LIN {X 0,Y 474.292,Z 613.364,A -85,B 0,C 180,E1 -7469.284,E2 -7469.284} C_VEL
LIN {X 0,Y 475.962,Z 468.165,A -85,B 0,C 180,E1 -7471.57,E2 -7471.57} C_VEL
LIN {X 0,Y 471.306,Z 449.007,A -85,B 0,C 180,E1 -7472.133,E2 -7472.133} C_VEL
LIN {X 0,Y 471.034,Z 448.055,A -85,B 0,C 180,E1 -7472.181,E2 -7472.181} C_VEL
LIN {X 0,Y 469.089,Z 439.057,A -85,B 0,C 180,E1 -7473.866,E2 -7473.866} C_VEL
LIN {X 0,Y 467.706,Z 432.847,A -85,B 0,C 180,E1 -7475.065,E2 -7475.065} C_VEL
LIN {X 0,Y 467.699,Z 432.856,A -85,B 0,C 180,E1 -7477.773,E2 -7477.773} C_VEL
LIN {X 0,Y 467.676,Z 432.847,A -85,B 0,C 180,E1 -7481.266,E2 -7481.266} C_VEL
LIN {X 0,Y 467.615,Z 432.864,A -85,B 0,C 180,E1 -7483.915,E2 -7483.915} C_VEL
LIN {X 0,Y 467.6,Z 432.861,A -85,B 0,C 180,E1 -7486.593,E2 -7486.593} C_VEL
LIN {X 0,Y 467.628,Z 432.861,A -85,B 0,C 180,E1 -7489.308,E2 -7489.308} C_VEL
LIN {X 0,Y 467.541,Z 432.872,A -85,B 0,C 180,E1 -7492.074,E2 -7492.074} C_VEL
LIN {X 0,Y 467.608,Z 432.856,A -85,B 0,C 180,E1 -7494.887,E2 -7494.887} C_VEL
LIN {X 0,Y 467.631,Z 432.857,A -85,B 0,C 180,E1 -7497.768,E2 -7497.768} C_VEL
LIN {X 0,Y 467.573,Z 432.865,A -85,B 0,C 180,E1 -7501.045,E2 -7501.045} C_VEL
LIN {X 0,Y 467.593,Z 432.863,A -85,B 0,C 180,E1 -7504.242,E2 -7504.242} C_VEL
LIN {X 0,Y 467.553,Z 432.866,A -85,B 0,C 180,E1 -7507.187,E2 -7507.187} C_VEL
LIN {X 0,Y 467.582,Z 432.863,A -85,B 0,C 180,E1 -7510.264,E2 -7510.264} C_VEL
LIN {X 0,Y 467.589,Z 432.858,A -85,B 0,C 180,E1 -7512.567,E2 -7512.567} C_VEL
LIN {X 0,Y 467.573,Z 432.863,A -85,B 0,C 180,E1 -7515.053,E2 -7515.053} C_VEL
LIN {X 0,Y 467.591,Z 432.866,A -85,B 0,C 180,E1 -7517.44,E2 -7517.44} C_VEL
LIN {X 0,Y 467.602,Z 432.86,A -85,B 0,C 180,E1 -7520.857,E2 -7520.857} C_VEL
LIN {X 0,Y 467.565,Z 432.86,A -85,B 0,C 180,E1 -7524.26,E2 -7524.26} C_VEL
LIN {X 0,Y 467.583,Z 432.865,A -85,B 0,C 180,E1 -7527.321,E2 -7527.321} C_VEL
LIN {X 0,Y 467.571,Z 432.857,A -85,B 0,C 180,E1 -7530.667,E2 -7530.667} C_VEL
LIN {X 0,Y 467.629,Z 432.858,A -85,B 0,C 180,E1 -7533.2,E2 -7533.2} C_VEL
LIN {X 0,Y 467.593,Z 432.852,A -85,B 0,C 180,E1 -7536.468,E2 -7536.468} C_VEL
LIN {X 0,Y 467.623,Z 432.863,A -85,B 0,C 180,E1 -7539.777,E2 -7539.777} C_VEL
LIN {X 0,Y 467.609,Z 432.853,A -85,B 0,C 180,E1 -7542.507,E2 -7542.507} C_VEL
LIN {X 0,Y 467.606,Z 432.857,A -85,B 0,C 180,E1 -7545.196,E2 -7545.196} C_VEL
LIN {X 0,Y 467.656,Z 432.855,A -85,B 0,C 180,E1 -7547.854,E2 -7547.854} C_VEL
LIN {X 0,Y 467.682,Z 432.845,A -85,B 0,C 180,E1 -7551.357,E2 -7551.357} C_VEL
LIN {X 0,Y 467.743,Z 432.845,A -85,B 0,C 180,E1 -7553.962,E2 -7553.962} C_VEL
LIN {X 0,Y 467.859,Z 432.824,A -85,B 0,C 180,E1 -7557.417,E2 -7557.417} C_VEL
LIN {X 0,Y 467.882,Z 432.829,A -85,B 0,C 180,E1 -7560,E2 -7560} C_VEL
LIN {X 0,Y 467.86,Z 432.824,A -85,B 0,C 180,E1 -7562.583,E2 -7562.583} C_VEL
LIN {X 0,Y 467.743,Z 432.843,A -85,B 0,C 180,E1 -7566.037,E2 -7566.037} C_VEL
LIN {X 0,Y 467.681,Z 432.849,A -85,B 0,C 180,E1 -7568.643,E2 -7568.643} C_VEL
LIN {X 0,Y 467.655,Z 432.848,A -85,B 0,C 180,E1 -7572.145,E2 -7572.145} C_VEL
LIN {X 0,Y 467.639,Z 432.862,A -85,B 0,C 180,E1 -7575.695,E2 -7575.695} C_VEL
LIN {X 0,Y 467.616,Z 432.849,A -85,B 0,C 180,E1 -7578.764,E2 -7578.764} C_VEL
LIN {X 0,Y 467.58,Z 432.864,A -85,B 0,C 180,E1 -7581.268,E2 -7581.268} C_VEL
LIN {X 0,Y 467.573,Z 432.868,A -85,B 0,C 180,E1 -7583.943,E2 -7583.943} C_VEL
LIN {X 0,Y 467.615,Z 432.858,A -85,B 0,C 180,E1 -7586.8,E2 -7586.8} C_VEL
LIN {X 0,Y 467.579,Z 432.87,A -85,B 0,C 180,E1 -7589.736,E2 -7589.736} C_VEL
LIN {X 0,Y 467.583,Z 432.862,A -85,B 0,C 180,E1 -7592.758,E2 -7592.758} C_VEL
LIN {X 0,Y 467.556,Z 432.871,A -85,B 0,C 180,E1 -7595.889,E2 -7595.889} C_VEL
LIN {X 0,Y 467.582,Z 432.864,A -85,B 0,C 180,E1 -7599.145,E2 -7599.145} C_VEL
LIN {X 0,Y 467.586,Z 432.862,A -85,B 0,C 180,E1 -7602.567,E2 -7602.567} C_VEL
LIN {X 0,Y 467.57,Z 432.865,A -85,B 0,C 180,E1 -7605.053,E2 -7605.053} C_VEL
LIN {X 0,Y 467.625,Z 432.862,A -85,B 0,C 180,E1 -7607.444,E2 -7607.444} C_VEL
LIN {X 0,Y 467.582,Z 432.864,A -85,B 0,C 180,E1 -7610.855,E2 -7610.855} C_VEL
LIN {X 0,Y 467.56,Z 432.871,A -85,B 0,C 180,E1 -7614.261,E2 -7614.261} C_VEL
LIN {X 0,Y 467.582,Z 432.869,A -85,B 0,C 180,E1 -7617.321,E2 -7617.321} C_VEL
LIN {X 0,Y 467.595,Z 432.887,A -85,B 0,C 180,E1 -7619.549,E2 -7619.549} C_VEL
LIN {X 0,Y 471.189,Z 447.756,A -85,B 0,C 180,E1 -7622.098,E2 -7622.098} C_VEL
LIN {X 0,Y 472.292,Z 452.989,A -85,B 0,C 180,E1 -7622.963,E2 -7622.963} C_VEL
LIN {X 0,Y 471.349,Z 470.678,A -85,B 0,C 180,E1 -7625.577,E2 -7625.577} C_VEL
LIN {X 0,Y 471.209,Z 472.852,A -85,B 0,C 180,E1 -7625.88,E2 -7625.88} C_VEL
LIN {X 0,Y 475.856,Z 496.892,A -85,B 0,C 180,E1 -7626.517,E2 -7626.517} C_VEL
LIN {X 0,Y 474.168,Z 638.503,A -85,B 0,C 180,E1 -7628.736,E2 -7628.736} C_VEL
LIN {X 0,Y 473.646,Z 654.003,A -85,B 0,C 180,E1 -7629.138,E2 -7629.138} C_VEL
LIN {X 0,Y 473.017,Z 668.829,A -85,B 0,C 180,E1 -7629.7,E2 -7629.7} C_VEL
LIN {X 0,Y 472.245,Z 683.472,A -85,B 0,C 180,E1 -7630.437,E2 -7630.437} C_VEL
LIN {X 0,Y 471.45,Z 697.08,A -85,B 0,C 180,E1 -7631.306,E2 -7631.306} C_VEL
LIN {X 0,Y 470.626,Z 709.613,A -85,B 0,C 180,E1 -7632.286,E2 -7632.286} C_VEL
LIN {X 0,Y 469.805,Z 722.347,A -85,B 0,C 180,E1 -7633.487,E2 -7633.487} C_VEL
LIN {X 0,Y 468.951,Z 733.908,A -85,B 0,C 180,E1 -7634.795,E2 -7634.795} C_VEL
LIN {X 0,Y 468.346,Z 743.643,A -85,B 0,C 180,E1 -7636.107,E2 -7636.107} C_VEL
LIN {X 0,Y 467.661,Z 753.221,A -85,B 0,C 180,E1 -7637.639,E2 -7637.639} C_VEL
LIN {X 0,Y 467.377,Z 761.161,A -85,B 0,C 180,E1 -7639.166,E2 -7639.166} C_VEL
LIN {X 0,Y 467.011,Z 768.591,A -85,B 0,C 180,E1 -7640.908,E2 -7640.908} C_VEL
LIN {X 0,Y 466.818,Z 774.485,A -85,B 0,C 180,E1 -7642.647,E2 -7642.647} C_VEL
LIN {X 0,Y 466.721,Z 777.986,A -85,B 0,C 180,E1 -7643.949,E2 -7643.949} C_VEL
LIN {X 0,Y 466.616,Z 781.525,A -85,B 0,C 180,E1 -7645.681,E2 -7645.681} C_VEL
LIN {X 0,Y 466.638,Z 783.854,A -85,B 0,C 180,E1 -7647.41,E2 -7647.41} C_VEL
LIN {X 0,Y 466.616,Z 785.022,A -85,B 0,C 180,E1 -7649.137,E2 -7649.137} C_VEL
LIN {X 0,Y 466.615,Z 785.016,A -85,B 0,C 180,E1 -7650.863,E2 -7650.863} C_VEL
LIN {X 0,Y 466.64,Z 783.835,A -85,B 0,C 180,E1 -7652.589,E2 -7652.589} C_VEL
LIN {X 0,Y 466.616,Z 781.496,A -85,B 0,C 180,E1 -7654.318,E2 -7654.318} C_VEL
LIN {X 0,Y 466.73,Z 777.954,A -85,B 0,C 180,E1 -7656.05,E2 -7656.05} C_VEL
LIN {X 0,Y 466.834,Z 773.112,A -85,B 0,C 180,E1 -7657.786,E2 -7657.786} C_VEL
LIN {X 0,Y 467.053,Z 766.845,A -85,B 0,C 180,E1 -7659.527,E2 -7659.527} C_VEL
LIN {X 0,Y 467.518,Z 758.98,A -85,B 0,C 180,E1 -7661.269,E2 -7661.269} C_VEL
LIN {X 0,Y 467.904,Z 750.519,A -85,B 0,C 180,E1 -7662.814,E2 -7662.814} C_VEL
LIN {X 0,Y 468.512,Z 740.532,A -85,B 0,C 180,E1 -7664.33,E2 -7664.33} C_VEL
LIN {X 0,Y 469.197,Z 730.234,A -85,B 0,C 180,E1 -7665.641,E2 -7665.641} C_VEL
LIN {X 0,Y 469.997,Z 718.835,A -85,B 0,C 180,E1 -7666.862,E2 -7666.862} C_VEL
LIN {X 0,Y 470.742,Z 706.933,A -85,B 0,C 180,E1 -7667.933,E2 -7667.933} C_VEL
LIN {X 0,Y 471.619,Z 693.812,A -85,B 0,C 180,E1 -7668.911,E2 -7668.911} C_VEL
LIN {X 0,Y 472.463,Z 679.406,A -85,B 0,C 180,E1 -7669.779,E2 -7669.779} C_VEL
LIN {X 0,Y 473.21,Z 665.055,A -85,B 0,C 180,E1 -7670.453,E2 -7670.453} C_VEL
LIN {X 0,Y 473.758,Z 650.356,A -85,B 0,C 180,E1 -7670.97,E2 -7670.97} C_VEL
LIN {X 0,Y 474.21,Z 635.624,A -85,B 0,C 180,E1 -7671.318,E2 -7671.318} C_VEL
LIN {X 0,Y 475.906,Z 497.322,A -85,B 0,C 180,E1 -7673.48,E2 -7673.48} C_VEL
LIN {X 0,Y 471.18,Z 472.312,A -85,B 0,C 180,E1 -7674.158,E2 -7674.158} C_VEL
LIN {X 0,Y 472.251,Z 452.84,A -85,B 0,C 180,E1 -7677.036,E2 -7677.036} C_VEL
LIN {X 0,Y 469.543,Z 440.542,A -85,B 0,C 180,E1 -7679.104,E2 -7679.104} C_VEL
LIN {X 0,Y 467.59,Z 432.868,A -85,B 0,C 180,E1 -7680.481,E2 -7680.481} C_VEL
LIN {X 0,Y 467.583,Z 432.865,A -85,B 0,C 180,E1 -7683.787,E2 -7683.787} C_VEL
LIN {X 0,Y 467.547,Z 432.867,A -85,B 0,C 180,E1 -7687.186,E2 -7687.186} C_VEL
LIN {X 0,Y 467.593,Z 432.863,A -85,B 0,C 180,E1 -7690.262,E2 -7690.262} C_VEL
LIN {X 0,Y 467.614,Z 432.859,A -85,B 0,C 180,E1 -7692.571,E2 -7692.571} C_VEL
LIN {X 0,Y 467.565,Z 432.867,A -85,B 0,C 180,E1 -7695.053,E2 -7695.053} C_VEL
LIN {X 0,Y 467.583,Z 432.861,A -85,B 0,C 180,E1 -7697.439,E2 -7697.439} C_VEL
LIN {X 0,Y 467.576,Z 432.866,A -85,B 0,C 180,E1 -7700.855,E2 -7700.855} C_VEL
LIN {X 0,Y 467.557,Z 432.87,A -85,B 0,C 180,E1 -7704.26,E2 -7704.26} C_VEL
LIN {X 0,Y 467.575,Z 432.861,A -85,B 0,C 180,E1 -7707.32,E2 -7707.32} C_VEL
LIN {X 0,Y 467.563,Z 432.869,A -85,B 0,C 180,E1 -7710.667,E2 -7710.667} C_VEL
LIN {X 0,Y 467.62,Z 432.855,A -85,B 0,C 180,E1 -7713.2,E2 -7713.2} C_VEL
LIN {X 0,Y 467.585,Z 432.865,A -85,B 0,C 180,E1 -7716.468,E2 -7716.468} C_VEL
LIN {X 0,Y 467.616,Z 432.857,A -85,B 0,C 180,E1 -7719.777,E2 -7719.777} C_VEL
LIN {X 0,Y 467.602,Z 432.861,A -85,B 0,C 180,E1 -7722.507,E2 -7722.507} C_VEL
LIN {X 0,Y 467.598,Z 432.86,A -85,B 0,C 180,E1 -7725.196,E2 -7725.196} C_VEL
LIN {X 0,Y 467.675,Z 432.851,A -85,B 0,C 180,E1 -7727.855,E2 -7727.855} C_VEL
LIN {X 0,Y 467.675,Z 432.85,A -85,B 0,C 180,E1 -7731.357,E2 -7731.357} C_VEL
LIN {X 0,Y 467.736,Z 432.845,A -85,B 0,C 180,E1 -7733.963,E2 -7733.963} C_VEL
LIN {X 0,Y 467.854,Z 432.826,A -85,B 0,C 180,E1 -7737.417,E2 -7737.417} C_VEL
LIN {X 0,Y 467.875,Z 432.829,A -85,B 0,C 180,E1 -7740,E2 -7740} C_VEL
LIN {X 0,Y 467.854,Z 432.834,A -85,B 0,C 180,E1 -7742.583,E2 -7742.583} C_VEL
LIN {X 0,Y 467.738,Z 432.845,A -85,B 0,C 180,E1 -7746.038,E2 -7746.038} C_VEL
LIN {X 0,Y 467.675,Z 432.856,A -85,B 0,C 180,E1 -7748.643,E2 -7748.643} C_VEL
LIN {X 0,Y 467.648,Z 432.857,A -85,B 0,C 180,E1 -7752.146,E2 -7752.146} C_VEL
LIN {X 0,Y 467.648,Z 432.855,A -85,B 0,C 180,E1 -7755.695,E2 -7755.695} C_VEL
LIN {X 0,Y 467.611,Z 432.862,A -85,B 0,C 180,E1 -7758.765,E2 -7758.765} C_VEL
LIN {X 0,Y 467.575,Z 432.863,A -85,B 0,C 180,E1 -7761.269,E2 -7761.269} C_VEL
LIN {X 0,Y 467.567,Z 432.868,A -85,B 0,C 180,E1 -7763.944,E2 -7763.944} C_VEL
LIN {X 0,Y 467.622,Z 432.86,A -85,B 0,C 180,E1 -7766.8,E2 -7766.8} C_VEL
LIN {X 0,Y 467.582,Z 432.863,A -85,B 0,C 180,E1 -7769.736,E2 -7769.736} C_VEL
LIN {X 0,Y 467.579,Z 432.865,A -85,B 0,C 180,E1 -7772.759,E2 -7772.759} C_VEL
LIN {X 0,Y 467.553,Z 432.871,A -85,B 0,C 180,E1 -7775.89,E2 -7775.89} C_VEL
LIN {X 0,Y 467.615,Z 432.865,A -85,B 0,C 180,E1 -7779.142,E2 -7779.142} C_VEL
LIN {X 0,Y 467.631,Z 432.96,A -85,B 0,C 180,E1 -7780.945,E2 -7780.945} C_VEL
LIN {X 0,Y 470.519,Z 445.746,A -85,B 0,C 180,E1 -7783.4,E2 -7783.4} C_VEL
LIN {X 0,Y 471.119,Z 448.459,A -85,B 0,C 180,E1 -7783.911,E2 -7783.911} C_VEL
LIN {X 0,Y 474.437,Z 461.432,A -85,B 0,C 180,E1 -7784.311,E2 -7784.311} C_VEL
LIN {X 0,Y 476.156,Z 469.425,A -85,B 0,C 180,E1 -7784.534,E2 -7784.534} C_VEL
LIN {X 0,Y 474.316,Z 613.801,A -85,B 0,C 180,E1 -7786.807,E2 -7786.807} C_VEL
LIN {X 0,Y 473.816,Z 629.451,A -85,B 0,C 180,E1 -7787.231,E2 -7787.231} C_VEL
LIN {X 0,Y 473.277,Z 643.627,A -85,B 0,C 180,E1 -7787.784,E2 -7787.784} C_VEL
LIN {X 0,Y 472.516,Z 658.62,A -85,B 0,C 180,E1 -7788.558,E2 -7788.558} C_VEL
LIN {X 0,Y 471.701,Z 672.281,A -85,B 0,C 180,E1 -7789.453,E2 -7789.453} C_VEL
LIN {X 0,Y 471.315,Z 678.799,A -85,B 0,C 180,E1 -7789.955,E2 -7789.955} C_VEL
LIN {X 0,Y 470.421,Z 683.716,A -85,B 0,C 180,E1 -7790.339,E2 -7790.339} C_VEL
LIN {X 0,Y 467.106,Z 691.605,A -85,B 0,C 180,E1 -7790.955,E2 -7790.955} C_VEL
LIN {X 0,Y 463.735,Z 699.161,A -85,B 0,C 180,E1 -7791.631,E2 -7791.631} C_VEL
LIN {X 0,Y 462.763,Z 703.515,A -85,B 0,C 180,E1 -7792.105,E2 -7792.105} C_VEL
LIN {X 0,Y 461.998,Z 713.096,A -85,B 0,C 180,E1 -7793.34,E2 -7793.34} C_VEL
LIN {X 0,Y 461.327,Z 722.98,A -85,B 0,C 180,E1 -7794.85,E2 -7794.85} C_VEL
LIN {X 0,Y 460.739,Z 731.593,A -85,B 0,C 180,E1 -7796.432,E2 -7796.432} C_VEL
LIN {X 0,Y 460.203,Z 739.522,A -85,B 0,C 180,E1 -7798.207,E2 -7798.207} C_VEL
LIN {X 0,Y 459.976,Z 745.004,A -85,B 0,C 180,E1 -7799.722,E2 -7799.722} C_VEL
LIN {X 0,Y 459.74,Z 749.421,A -85,B 0,C 180,E1 -7801.215,E2 -7801.215} C_VEL
LIN {X 0,Y 459.622,Z 752.795,A -85,B 0,C 180,E1 -7802.696,E2 -7802.696} C_VEL
LIN {X 0,Y 459.459,Z 755.962,A -85,B 0,C 180,E1 -7804.641,E2 -7804.641} C_VEL
LIN {X 0,Y 459.411,Z 757.715,A -85,B 0,C 180,E1 -7806.617,E2 -7806.617} C_VEL
LIN {X 0,Y 459.389,Z 758.052,A -85,B 0,C 180,E1 -7808.46,E2 -7808.46} C_VEL
LIN {X 0,Y 459.447,Z 757.117,A -85,B 0,C 180,E1 -7810.335,E2 -7810.335} C_VEL
LIN {X 0,Y 459.533,Z 754.911,A -85,B 0,C 180,E1 -7812.19,E2 -7812.19} C_VEL
LIN {X 0,Y 459.715,Z 751.415,A -85,B 0,C 180,E1 -7814.028,E2 -7814.028} C_VEL
LIN {X 0,Y 459.88,Z 746.602,A -85,B 0,C 180,E1 -7815.847,E2 -7815.847} C_VEL
LIN {X 0,Y 460.206,Z 740.359,A -85,B 0,C 180,E1 -7817.656,E2 -7817.656} C_VEL
LIN {X 0,Y 460.66,Z 732.532,A -85,B 0,C 180,E1 -7819.452,E2 -7819.452} C_VEL
LIN {X 0,Y 461.197,Z 724.229,A -85,B 0,C 180,E1 -7821.014,E2 -7821.014} C_VEL
LIN {X 0,Y 461.921,Z 714.254,A -85,B 0,C 180,E1 -7822.57,E2 -7822.57} C_VEL
LIN {X 0,Y 462.671,Z 704.091,A -85,B 0,C 180,E1 -7823.897,E2 -7823.897} C_VEL
LIN {X 0,Y 463.549,Z 692.016,A -85,B 0,C 180,E1 -7825.217,E2 -7825.217} C_VEL
LIN {X 0,Y 464.521,Z 678.617,A -85,B 0,C 180,E1 -7826.422,E2 -7826.422} C_VEL
LIN {X 0,Y 465.415,Z 665.239,A -85,B 0,C 180,E1 -7827.404,E2 -7827.404} C_VEL
LIN {X 0,Y 466.207,Z 651.434,A -85,B 0,C 180,E1 -7828.219,E2 -7828.219} C_VEL
LIN {X 0,Y 466.911,Z 636.009,A -85,B 0,C 180,E1 -7828.922,E2 -7828.922} C_VEL
LIN {X 0,Y 467.471,Z 620.257,A -85,B 0,C 180,E1 -7829.435,E2 -7829.435} C_VEL
LIN {X 0,Y 467.799,Z 604.734,A -85,B 0,C 180,E1 -7829.758,E2 -7829.758} C_VEL
LIN {X 0,Y 469.488,Z 469.443,A -85,B 0,C 180,E1 -7831.893,E2 -7831.893} C_VEL
LIN {X 0,Y 465.042,Z 451.21,A -85,B 0,C 180,E1 -7832.441,E2 -7832.441} C_VEL
LIN {X 0,Y 463.945,Z 448.293,A -85,B 0,C 180,E1 -7832.565,E2 -7832.565} C_VEL
LIN {X 0,Y 460.678,Z 433.722,A -85,B 0,C 180,E1 -7835.389,E2 -7835.389} C_VEL
LIN {X 0,Y 460.671,Z 433.73,A -85,B 0,C 180,E1 -7837.892,E2 -7837.892} C_VEL
LIN {X 0,Y 460.635,Z 433.726,A -85,B 0,C 180,E1 -7841.44,E2 -7841.44} C_VEL
LIN {X 0,Y 460.559,Z 433.741,A -85,B 0,C 180,E1 -7844.132,E2 -7844.132} C_VEL
LIN {X 0,Y 460.568,Z 433.738,A -85,B 0,C 180,E1 -7846.854,E2 -7846.854} C_VEL
LIN {X 0,Y 460.573,Z 433.744,A -85,B 0,C 180,E1 -7849.616,E2 -7849.616} C_VEL
LIN {X 0,Y 460.517,Z 433.744,A -85,B 0,C 180,E1 -7852.429,E2 -7852.429} C_VEL
LIN {X 0,Y 460.572,Z 433.742,A -85,B 0,C 180,E1 -7855.802,E2 -7855.802} C_VEL
LIN {X 0,Y 460.559,Z 433.735,A -85,B 0,C 180,E1 -7858.233,E2 -7858.233} C_VEL
LIN {X 0,Y 460.526,Z 433.745,A -85,B 0,C 180,E1 -7861.283,E2 -7861.283} C_VEL
LIN {X 0,Y 460.537,Z 433.74,A -85,B 0,C 180,E1 -7864.506,E2 -7864.506} C_VEL
LIN {X 0,Y 460.531,Z 433.739,A -85,B 0,C 180,E1 -7867.62,E2 -7867.62} C_VEL
LIN {X 0,Y 460.546,Z 433.74,A -85,B 0,C 180,E1 -7870.269,E2 -7870.269} C_VEL
LIN {X 0,Y 460.511,Z 433.743,A -85,B 0,C 180,E1 -7873.374,E2 -7873.374} C_VEL
LIN {X 0,Y 460.502,Z 433.743,A -85,B 0,C 180,E1 -7876.624,E2 -7876.624} C_VEL
LIN {X 0,Y 460.56,Z 433.741,A -85,B 0,C 180,E1 -7879.728,E2 -7879.728} C_VEL
LIN {X 0,Y 460.53,Z 433.738,A -85,B 0,C 180,E1 -7882.519,E2 -7882.519} C_VEL
LIN {X 0,Y 460.551,Z 433.741,A -85,B 0,C 180,E1 -7885.624,E2 -7885.624} C_VEL
LIN {X 0,Y 460.538,Z 433.737,A -85,B 0,C 180,E1 -7888.744,E2 -7888.744} C_VEL
LIN {X 0,Y 460.59,Z 433.734,A -85,B 0,C 180,E1 -7892.252,E2 -7892.252} C_VEL
LIN {X 0,Y 460.56,Z 433.735,A -85,B 0,C 180,E1 -7894.705,E2 -7894.705} C_VEL
LIN {X 0,Y 460.511,Z 433.74,A -85,B 0,C 180,E1 -7897.571,E2 -7897.571} C_VEL
LIN {X 0,Y 460.569,Z 433.736,A -85,B 0,C 180,E1 -7900.384,E2 -7900.384} C_VEL
LIN {X 0,Y 460.566,Z 433.731,A -85,B 0,C 180,E1 -7903.146,E2 -7903.146} C_VEL
LIN {X 0,Y 460.555,Z 433.742,A -85,B 0,C 180,E1 -7905.868,E2 -7905.868} C_VEL
LIN {X 0,Y 460.611,Z 433.727,A -85,B 0,C 180,E1 -7908.559,E2 -7908.559} C_VEL
LIN {X 0,Y 460.695,Z 433.721,A -85,B 0,C 180,E1 -7912.108,E2 -7912.108} C_VEL
LIN {X 0,Y 460.697,Z 433.718,A -85,B 0,C 180,E1 -7914.748,E2 -7914.748} C_VEL
LIN {X 0,Y 460.8,Z 433.703,A -85,B 0,C 180,E1 -7917.377,E2 -7917.377} C_VEL
LIN {X 0,Y 460.853,Z 433.704,A -85,B 0,C 180,E1 -7920,E2 -7920} C_VEL
LIN {X 0,Y 460.824,Z 433.7,A -85,B 0,C 180,E1 -7922.622,E2 -7922.622} C_VEL
LIN {X 0,Y 460.709,Z 433.718,A -85,B 0,C 180,E1 -7926.13,E2 -7926.13} C_VEL
LIN {X 0,Y 460.628,Z 433.728,A -85,B 0,C 180,E1 -7928.776,E2 -7928.776} C_VEL
LIN {X 0,Y 460.613,Z 433.723,A -85,B 0,C 180,E1 -7932.445,E2 -7932.445} C_VEL
LIN {X 0,Y 460.599,Z 433.735,A -85,B 0,C 180,E1 -7935.997,E2 -7935.997} C_VEL
LIN {X 0,Y 460.57,Z 433.727,A -85,B 0,C 180,E1 -7938.902,E2 -7938.902} C_VEL
LIN {X 0,Y 460.515,Z 433.747,A -85,B 0,C 180,E1 -7941.485,E2 -7941.485} C_VEL
LIN {X 0,Y 460.542,Z 433.74,A -85,B 0,C 180,E1 -7944.332,E2 -7944.332} C_VEL
LIN {X 0,Y 460.578,Z 433.737,A -85,B 0,C 180,E1 -7947.243,E2 -7947.243} C_VEL
LIN {X 0,Y 460.521,Z 433.742,A -85,B 0,C 180,E1 -7950.239,E2 -7950.239} C_VEL
LIN {X 0,Y 460.529,Z 433.744,A -85,B 0,C 180,E1 -7953.325,E2 -7953.325} C_VEL
LIN {X 0,Y 460.479,Z 433.747,A -85,B 0,C 180,E1 -7956.529,E2 -7956.529} C_VEL
LIN {X 0,Y 460.557,Z 433.742,A -85,B 0,C 180,E1 -7959.86,E2 -7959.86} C_VEL
LIN {X 0,Y 460.513,Z 433.743,A -85,B 0,C 180,E1 -7962.9,E2 -7962.9} C_VEL
LIN {X 0,Y 460.524,Z 433.747,A -85,B 0,C 180,E1 -7965.829,E2 -7965.829} C_VEL
LIN {X 0,Y 460.535,Z 433.742,A -85,B 0,C 180,E1 -7968.989,E2 -7968.989} C_VEL
LIN {X 0,Y 460.526,Z 433.745,A -85,B 0,C 180,E1 -7971.267,E2 -7971.267} C_VEL
LIN {X 0,Y 460.51,Z 433.748,A -85,B 0,C 180,E1 -7974.554,E2 -7974.554} C_VEL
LIN {X 0,Y 460.532,Z 433.744,A -85,B 0,C 180,E1 -7977.715,E2 -7977.715} C_VEL
LIN {X 0,Y 460.548,Z 433.832,A -85,B 0,C 180,E1 -7979.223,E2 -7979.223} C_VEL
LIN {X 0,Y 464.059,Z 448.047,A -85,B 0,C 180,E1 -7981.713,E2 -7981.713} C_VEL
LIN {X 0,Y 465.493,Z 454.798,A -85,B 0,C 180,E1 -7982.849,E2 -7982.849} C_VEL
LIN {X 0,Y 464.454,Z 472.525,A -85,B 0,C 180,E1 -7985.505,E2 -7985.505} C_VEL
LIN {X 0,Y 469.309,Z 497.459,A -85,B 0,C 180,E1 -7986.184,E2 -7986.184} C_VEL
LIN {X 0,Y 467.541,Z 638.122,A -85,B 0,C 180,E1 -7988.419,E2 -7988.419} C_VEL
LIN {X 0,Y 466.99,Z 653.689,A -85,B 0,C 180,E1 -7988.826,E2 -7988.826} C_VEL
LIN {X 0,Y 466.321,Z 669.079,A -85,B 0,C 180,E1 -7989.419,E2 -7989.419} C_VEL
LIN {X 0,Y 465.537,Z 683.208,A -85,B 0,C 180,E1 -7990.143,E2 -7990.143} C_VEL
LIN {X 0,Y 464.674,Z 696.828,A -85,B 0,C 180,E1 -7991.023,E2 -7991.023} C_VEL
LIN {X 0,Y 463.73,Z 710.667,A -85,B 0,C 180,E1 -7992.127,E2 -7992.127} C_VEL
LIN {X 0,Y 462.858,Z 723.186,A -85,B 0,C 180,E1 -7993.345,E2 -7993.345} C_VEL
LIN {X 0,Y 462.047,Z 733.678,A -85,B 0,C 180,E1 -7994.562,E2 -7994.562} C_VEL
LIN {X 0,Y 461.38,Z 743.417,A -85,B 0,C 180,E1 -7995.893,E2 -7995.893} C_VEL
LIN {X 0,Y 460.783,Z 751.983,A -85,B 0,C 180,E1 -7997.267,E2 -7997.267} C_VEL
LIN {X 0,Y 460.444,Z 759.928,A -85,B 0,C 180,E1 -7998.778,E2 -7998.778} C_VEL
LIN {X 0,Y 459.979,Z 766.687,A -85,B 0,C 180,E1 -8000.324,E2 -8000.324} C_VEL
LIN {X 0,Y 459.776,Z 772.941,A -85,B 0,C 180,E1 -8002.092,E2 -8002.092} C_VEL
LIN {X 0,Y 459.637,Z 777.777,A -85,B 0,C 180,E1 -8003.855,E2 -8003.855} C_VEL
LIN {X 0,Y 459.533,Z 781.317,A -85,B 0,C 180,E1 -8005.614,E2 -8005.614} C_VEL
LIN {X 0,Y 459.56,Z 783.647,A -85,B 0,C 180,E1 -8007.37,E2 -8007.37} C_VEL
LIN {X 0,Y 459.519,Z 784.815,A -85,B 0,C 180,E1 -8009.123,E2 -8009.123} C_VEL
LIN {X 0,Y 459.518,Z 784.809,A -85,B 0,C 180,E1 -8010.876,E2 -8010.876} C_VEL
LIN {X 0,Y 459.563,Z 783.627,A -85,B 0,C 180,E1 -8012.629,E2 -8012.629} C_VEL
LIN {X 0,Y 459.532,Z 781.287,A -85,B 0,C 180,E1 -8014.385,E2 -8014.385} C_VEL
LIN {X 0,Y 459.639,Z 777.742,A -85,B 0,C 180,E1 -8016.144,E2 -8016.144} C_VEL
LIN {X 0,Y 459.775,Z 772.9,A -85,B 0,C 180,E1 -8017.907,E2 -8017.907} C_VEL
LIN {X 0,Y 459.978,Z 766.629,A -85,B 0,C 180,E1 -8019.675,E2 -8019.675} C_VEL
LIN {X 0,Y 460.459,Z 758.761,A -85,B 0,C 180,E1 -8021.444,E2 -8021.444} C_VEL
LIN {X 0,Y 460.898,Z 750.525,A -85,B 0,C 180,E1 -8022.975,E2 -8022.975} C_VEL
LIN {X 0,Y 461.573,Z 740.309,A -85,B 0,C 180,E1 -8024.55,E2 -8024.55} C_VEL
LIN {X 0,Y 462.313,Z 730.008,A -85,B 0,C 180,E1 -8025.88,E2 -8025.88} C_VEL
LIN {X 0,Y 463.236,Z 717.683,A -85,B 0,C 180,E1 -8027.212,E2 -8027.212} C_VEL
LIN {X 0,Y 464.067,Z 705.402,A -85,B 0,C 180,E1 -8028.315,E2 -8028.315} C_VEL
LIN {X 0,Y 464.977,Z 691.994,A -85,B 0,C 180,E1 -8029.307,E2 -8029.307} C_VEL
LIN {X 0,Y 465.905,Z 677.195,A -85,B 0,C 180,E1 -8030.185,E2 -8030.185} C_VEL
LIN {X 0,Y 466.637,Z 662.471,A -85,B 0,C 180,E1 -8030.86,E2 -8030.86} C_VEL
LIN {X 0,Y 467.271,Z 647.421,A -85,B 0,C 180,E1 -8031.361,E2 -8031.361} C_VEL
LIN {X 0,Y 467.674,Z 632.474,A -85,B 0,C 180,E1 -8031.689,E2 -8031.689} C_VEL
LIN {X 0,Y 469.36,Z 497.451,A -85,B 0,C 180,E1 -8033.824,E2 -8033.824} C_VEL
LIN {X 0,Y 464.455,Z 472.084,A -85,B 0,C 180,E1 -8034.536,E2 -8034.536} C_VEL
LIN {X 0,Y 465.432,Z 454.521,A -85,B 0,C 180,E1 -8037.178,E2 -8037.178} C_VEL
LIN {X 0,Y 462.709,Z 442.309,A -85,B 0,C 180,E1 -8039.269,E2 -8039.269} C_VEL
LIN {X 0,Y 460.532,Z 433.747,A -85,B 0,C 180,E1 -8040.808,E2 -8040.808} C_VEL
LIN {X 0,Y 460.526,Z 433.744,A -85,B 0,C 180,E1 -8043.324,E2 -8043.324} C_VEL
LIN {X 0,Y 460.475,Z 433.753,A -85,B 0,C 180,E1 -8046.528,E2 -8046.528} C_VEL
LIN {X 0,Y 460.574,Z 433.737,A -85,B 0,C 180,E1 -8049.857,E2 -8049.857} C_VEL
LIN {X 0,Y 460.537,Z 433.738,A -85,B 0,C 180,E1 -8052.904,E2 -8052.904} C_VEL
LIN {X 0,Y 460.505,Z 433.749,A -85,B 0,C 180,E1 -8055.83,E2 -8055.83} C_VEL
LIN {X 0,Y 460.525,Z 433.743,A -85,B 0,C 180,E1 -8058.988,E2 -8058.988} C_VEL
LIN {X 0,Y 460.52,Z 433.743,A -85,B 0,C 180,E1 -8061.267,E2 -8061.267} C_VEL
LIN {X 0,Y 460.507,Z 433.748,A -85,B 0,C 180,E1 -8064.554,E2 -8064.554} C_VEL
LIN {X 0,Y 460.525,Z 433.741,A -85,B 0,C 180,E1 -8067.715,E2 -8067.715} C_VEL
LIN {X 0,Y 460.533,Z 433.744,A -85,B 0,C 180,E1 -8070.769,E2 -8070.769} C_VEL
LIN {X 0,Y 460.561,Z 433.736,A -85,B 0,C 180,E1 -8073.735,E2 -8073.735} C_VEL
LIN {X 0,Y 460.539,Z 433.744,A -85,B 0,C 180,E1 -8076.624,E2 -8076.624} C_VEL
LIN {X 0,Y 460.544,Z 433.736,A -85,B 0,C 180,E1 -8079.453,E2 -8079.453} C_VEL
LIN {X 0,Y 460.552,Z 433.743,A -85,B 0,C 180,E1 -8082.23,E2 -8082.23} C_VEL
LIN {X 0,Y 460.557,Z 433.738,A -85,B 0,C 180,E1 -8084.965,E2 -8084.965} C_VEL
LIN {X 0,Y 460.622,Z 433.728,A -85,B 0,C 180,E1 -8087.666,E2 -8087.666} C_VEL
LIN {X 0,Y 460.622,Z 433.728,A -85,B 0,C 180,E1 -8091.224,E2 -8091.224} C_VEL
LIN {X 0,Y 460.702,Z 433.72,A -85,B 0,C 180,E1 -8093.87,E2 -8093.87} C_VEL
LIN {X 0,Y 460.819,Z 433.702,A -85,B 0,C 180,E1 -8097.378,E2 -8097.378} C_VEL
LIN {X 0,Y 460.845,Z 433.705,A -85,B 0,C 180,E1 -8100,E2 -8100} C_VEL
LIN {X 0,Y 460.819,Z 433.71,A -85,B 0,C 180,E1 -8102.623,E2 -8102.623} C_VEL
LIN {X 0,Y 460.704,Z 433.722,A -85,B 0,C 180,E1 -8106.13,E2 -8106.13} C_VEL
LIN {X 0,Y 460.622,Z 433.733,A -85,B 0,C 180,E1 -8108.776,E2 -8108.776} C_VEL
LIN {X 0,Y 460.606,Z 433.739,A -85,B 0,C 180,E1 -8112.445,E2 -8112.445} C_VEL
LIN {X 0,Y 460.615,Z 433.734,A -85,B 0,C 180,E1 -8116.008,E2 -8116.008} C_VEL
LIN {X 0,Y 460.563,Z 433.737,A -85,B 0,C 180,E1 -8119.616,E2 -8119.616} C_VEL
LIN {X 0,Y 460.505,Z 433.752,A -85,B 0,C 180,E1 -8122.429,E2 -8122.429} C_VEL
LIN {X 0,Y 460.563,Z 433.74,A -85,B 0,C 180,E1 -8125.803,E2 -8125.803} C_VEL
LIN {X 0,Y 460.553,Z 433.745,A -85,B 0,C 180,E1 -8128.233,E2 -8128.233} C_VEL
LIN {X 0,Y 460.52,Z 433.744,A -85,B 0,C 180,E1 -8131.285,E2 -8131.285} C_VEL
LIN {X 0,Y 460.53,Z 433.745,A -85,B 0,C 180,E1 -8134.507,E2 -8134.507} C_VEL
LIN {X 0,Y 460.527,Z 433.746,A -85,B 0,C 180,E1 -8137.621,E2 -8137.621} C_VEL
LIN {X 0,Y 460.567,Z 433.805,A -85,B 0,C 180,E1 -8140.602,E2 -8140.602} C_VEL
LIN {X 0,Y 463.443,Z 446.216,A -85,B 0,C 180,E1 -8143.033,E2 -8143.033} C_VEL
LIN {X 0,Y 463.962,Z 448.732,A -85,B 0,C 180,E1 -8143.513,E2 -8143.513} C_VEL
LIN {X 0,Y 466.156,Z 454.96,A -85,B 0,C 180,E1 -8143.744,E2 -8143.744} C_VEL
LIN {X 0,Y 469.604,Z 469.923,A -85,B 0,C 180,E1 -8144.188,E2 -8144.188} C_VEL
LIN {X 0,Y 467.734,Z 613.627,A -85,B 0,C 180,E1 -8146.482,E2 -8146.482} C_VEL
LIN {X 0,Y 467.234,Z 629.203,A -85,B 0,C 180,E1 -8146.905,E2 -8146.905} C_VEL
LIN {X 0,Y 466.594,Z 644.62,A -85,B 0,C 180,E1 -8147.518,E2 -8147.518} C_VEL
LIN {X 0,Y 465.82,Z 658.855,A -85,B 0,C 180,E1 -8148.267,E2 -8148.267} C_VEL
LIN {X 0,Y 464.972,Z 672.601,A -85,B 0,C 180,E1 -8149.182,E2 -8149.182} C_VEL
LIN {X 0,Y 464.091,Z 685.353,A -85,B 0,C 180,E1 -8150.223,E2 -8150.223} C_VEL
LIN {X 0,Y 463.227,Z 697.249,A -85,B 0,C 180,E1 -8151.397,E2 -8151.397} C_VEL
LIN {X 0,Y 462.763,Z 703.515,A -85,B 0,C 180,E1 -8152.105,E2 -8152.105} C_VEL
LIN {X 0,Y 461.824,Z 707.77,A -85,B 0,C 180,E1 -8152.6,E2 -8152.6} C_VEL
LIN {X 0,Y 458.551,Z 714.532,A -85,B 0,C 180,E1 -8153.406,E2 -8153.406} C_VEL
LIN {X 0,Y 455.243,Z 720.853,A -85,B 0,C 180,E1 -8154.27,E2 -8154.27} C_VEL
LIN {X 0,Y 454.264,Z 724.419,A -85,B 0,C 180,E1 -8154.852,E2 -8154.852} C_VEL
LIN {X 0,Y 453.68,Z 733.014,A -85,B 0,C 180,E1 -8156.496,E2 -8156.496} C_VEL
LIN {X 0,Y 453.166,Z 740.231,A -85,B 0,C 180,E1 -8158.178,E2 -8158.178} C_VEL
LIN {X 0,Y 452.917,Z 745.604,A -85,B 0,C 180,E1 -8159.715,E2 -8159.715} C_VEL
LIN {X 0,Y 452.649,Z 749.938,A -85,B 0,C 180,E1 -8161.229,E2 -8161.229} C_VEL
LIN {X 0,Y 452.448,Z 754.173,A -85,B 0,C 180,E1 -8163.227,E2 -8163.227} C_VEL
LIN {X 0,Y 452.32,Z 756.88,A -85,B 0,C 180,E1 -8165.197,E2 -8165.197} C_VEL
LIN {X 0,Y 452.29,Z 758.179,A -85,B 0,C 180,E1 -8167.142,E2 -8167.142} C_VEL
LIN {X 0,Y 452.34,Z 758.139,A -85,B 0,C 180,E1 -8169.063,E2 -8169.063} C_VEL
LIN {X 0,Y 452.359,Z 756.798,A -85,B 0,C 180,E1 -8170.959,E2 -8170.959} C_VEL
LIN {X 0,Y 452.467,Z 754.173,A -85,B 0,C 180,E1 -8172.836,E2 -8172.836} C_VEL
LIN {X 0,Y 452.695,Z 750.249,A -85,B 0,C 180,E1 -8174.698,E2 -8174.698} C_VEL
LIN {X 0,Y 452.901,Z 744.997,A -85,B 0,C 180,E1 -8176.541,E2 -8176.541} C_VEL
LIN {X 0,Y 453.205,Z 739.626,A -85,B 0,C 180,E1 -8178.038,E2 -8178.038} C_VEL
LIN {X 0,Y 453.66,Z 732.191,A -85,B 0,C 180,E1 -8179.738,E2 -8179.738} C_VEL
LIN {X 0,Y 454.305,Z 723.67,A -85,B 0,C 180,E1 -8181.34,E2 -8181.34} C_VEL
LIN {X 0,Y 455.064,Z 713.656,A -85,B 0,C 180,E1 -8182.903,E2 -8182.903} C_VEL
LIN {X 0,Y 455.879,Z 703.37,A -85,B 0,C 180,E1 -8184.25,E2 -8184.25} C_VEL
LIN {X 0,Y 456.845,Z 691.066,A -85,B 0,C 180,E1 -8185.589,E2 -8185.589} C_VEL
LIN {X 0,Y 457.797,Z 678.144,A -85,B 0,C 180,E1 -8186.752,E2 -8186.752} C_VEL
LIN {X 0,Y 458.712,Z 665.396,A -85,B 0,C 180,E1 -8187.696,E2 -8187.696} C_VEL
LIN {X 0,Y 459.538,Z 651.573,A -85,B 0,C 180,E1 -8188.522,E2 -8188.522} C_VEL
LIN {X 0,Y 460.23,Z 637.433,A -85,B 0,C 180,E1 -8189.18,E2 -8189.18} C_VEL
LIN {X 0,Y 460.806,Z 622.279,A -85,B 0,C 180,E1 -8189.7,E2 -8189.7} C_VEL
LIN {X 0,Y 461.172,Z 606.382,A -85,B 0,C 180,E1 -8190.055,E2 -8190.055} C_VEL
LIN {X 0,Y 463.026,Z 470.802,A -85,B 0,C 180,E1 -8192.223,E2 -8192.223} C_VEL
LIN {X 0,Y 459.032,Z 454.277,A -85,B 0,C 180,E1 -8192.728,E2 -8192.728} C_VEL
LIN {X 0,Y 456.814,Z 448.521,A -85,B 0,C 180,E1 -8192.961,E2 -8192.961} C_VEL
LIN {X 0,Y 453.647,Z 434.599,A -85,B 0,C 180,E1 -8195.724,E2 -8195.724} C_VEL
LIN {X 0,Y 453.597,Z 434.609,A -85,B 0,C 180,E1 -8198.914,E2 -8198.914} C_VEL
LIN {X 0,Y 453.606,Z 434.607,A -85,B 0,C 180,E1 -8202.551,E2 -8202.551} C_VEL
LIN {X 0,Y 453.549,Z 434.613,A -85,B 0,C 180,E1 -8206.196,E2 -8206.196} C_VEL
LIN {X 0,Y 453.524,Z 434.615,A -85,B 0,C 180,E1 -8209.041,E2 -8209.041} C_VEL
LIN {X 0,Y 453.481,Z 434.625,A -85,B 0,C 180,E1 -8211.836,E2 -8211.836} C_VEL
LIN {X 0,Y 453.518,Z 434.611,A -85,B 0,C 180,E1 -8214.734,E2 -8214.734} C_VEL
LIN {X 0,Y 453.541,Z 434.61,A -85,B 0,C 180,E1 -8217.961,E2 -8217.961} C_VEL
LIN {X 0,Y 453.485,Z 434.619,A -85,B 0,C 180,E1 -8220.759,E2 -8220.759} C_VEL
LIN {X 0,Y 453.481,Z 434.624,A -85,B 0,C 180,E1 -8223.912,E2 -8223.912} C_VEL
LIN {X 0,Y 453.473,Z 434.62,A -85,B 0,C 180,E1 -8227.188,E2 -8227.188} C_VEL
LIN {X 0,Y 453.52,Z 434.613,A -85,B 0,C 180,E1 -8229.447,E2 -8229.447} C_VEL
LIN {X 0,Y 453.47,Z 434.617,A -85,B 0,C 180,E1 -8232.994,E2 -8232.994} C_VEL
LIN {X 0,Y 453.468,Z 434.626,A -85,B 0,C 180,E1 -8235.779,E2 -8235.779} C_VEL
LIN {X 0,Y 453.518,Z 434.612,A -85,B 0,C 180,E1 -8239.405,E2 -8239.405} C_VEL
LIN {X 0,Y 453.478,Z 434.618,A -85,B 0,C 180,E1 -8242.223,E2 -8242.223} C_VEL
LIN {X 0,Y 453.491,Z 434.614,A -85,B 0,C 180,E1 -8245.222,E2 -8245.222} C_VEL
LIN {X 0,Y 453.467,Z 434.618,A -85,B 0,C 180,E1 -8248.475,E2 -8248.475} C_VEL
LIN {X 0,Y 453.539,Z 434.614,A -85,B 0,C 180,E1 -8252.039,E2 -8252.039} C_VEL
LIN {X 0,Y 453.514,Z 434.616,A -85,B 0,C 180,E1 -8255.265,E2 -8255.265} C_VEL
LIN {X 0,Y 453.481,Z 434.617,A -85,B 0,C 180,E1 -8258.415,E2 -8258.415} C_VEL
LIN {X 0,Y 453.522,Z 434.614,A -85,B 0,C 180,E1 -8261.008,E2 -8261.008} C_VEL
LIN {X 0,Y 453.569,Z 434.605,A -85,B 0,C 180,E1 -8263.879,E2 -8263.879} C_VEL
LIN {X 0,Y 453.564,Z 434.613,A -85,B 0,C 180,E1 -8267.471,E2 -8267.471} C_VEL
LIN {X 0,Y 453.592,Z 434.597,A -85,B 0,C 180,E1 -8271.086,E2 -8271.086} C_VEL
LIN {X 0,Y 453.677,Z 434.6,A -85,B 0,C 180,E1 -8273.774,E2 -8273.774} C_VEL
LIN {X 0,Y 453.744,Z 434.581,A -85,B 0,C 180,E1 -8277.336,E2 -8277.336} C_VEL
LIN {X 0,Y 453.823,Z 434.58,A -85,B 0,C 180,E1 -8280,E2 -8280} C_VEL
LIN {X 0,Y 453.765,Z 434.579,A -85,B 0,C 180,E1 -8282.663,E2 -8282.663} C_VEL
LIN {X 0,Y 453.677,Z 434.593,A -85,B 0,C 180,E1 -8286.225,E2 -8286.225} C_VEL
LIN {X 0,Y 453.592,Z 434.605,A -85,B 0,C 180,E1 -8288.913,E2 -8288.913} C_VEL
LIN {X 0,Y 453.563,Z 434.601,A -85,B 0,C 180,E1 -8292.529,E2 -8292.529} C_VEL
LIN {X 0,Y 453.544,Z 434.611,A -85,B 0,C 180,E1 -8296.196,E2 -8296.196} C_VEL
LIN {X 0,Y 453.519,Z 434.605,A -85,B 0,C 180,E1 -8299.04,E2 -8299.04} C_VEL
LIN {X 0,Y 453.476,Z 434.625,A -85,B 0,C 180,E1 -8301.836,E2 -8301.836} C_VEL
LIN {X 0,Y 453.514,Z 434.615,A -85,B 0,C 180,E1 -8304.734,E2 -8304.734} C_VEL
LIN {X 0,Y 453.537,Z 434.615,A -85,B 0,C 180,E1 -8307.961,E2 -8307.961} C_VEL
LIN {X 0,Y 453.48,Z 434.617,A -85,B 0,C 180,E1 -8310.759,E2 -8310.759} C_VEL
LIN {X 0,Y 453.478,Z 434.625,A -85,B 0,C 180,E1 -8313.912,E2 -8313.912} C_VEL
LIN {X 0,Y 453.47,Z 434.622,A -85,B 0,C 180,E1 -8317.188,E2 -8317.188} C_VEL
LIN {X 0,Y 453.516,Z 434.619,A -85,B 0,C 180,E1 -8319.447,E2 -8319.447} C_VEL
LIN {X 0,Y 453.463,Z 434.622,A -85,B 0,C 180,E1 -8322.995,E2 -8322.995} C_VEL
LIN {X 0,Y 453.477,Z 434.625,A -85,B 0,C 180,E1 -8325.78,E2 -8325.78} C_VEL
LIN {X 0,Y 453.494,Z 434.621,A -85,B 0,C 180,E1 -8328.211,E2 -8328.211} C_VEL
LIN {X 0,Y 453.464,Z 434.627,A -85,B 0,C 180,E1 -8331.688,E2 -8331.688} C_VEL
LIN {X 0,Y 453.487,Z 434.624,A -85,B 0,C 180,E1 -8335.223,E2 -8335.223} C_VEL
LIN {X 0,Y 453.466,Z 434.626,A -85,B 0,C 180,E1 -8338.475,E2 -8338.475} C_VEL
LIN {X 0,Y 453.513,Z 434.688,A -85,B 0,C 180,E1 -8338.875,E2 -8338.875} C_VEL
LIN {X 0,Y 457.191,Z 449.64,A -85,B 0,C 180,E1 -8341.54,E2 -8341.54} C_VEL
LIN {X 0,Y 458.676,Z 456.462,A -85,B 0,C 180,E1 -8342.71,E2 -8342.71} C_VEL
LIN {X 0,Y 457.707,Z 472.291,A -85,B 0,C 180,E1 -8345.119,E2 -8345.119} C_VEL
LIN {X 0,Y 462.788,Z 499.008,A -85,B 0,C 180,E1 -8345.862,E2 -8345.862} C_VEL
LIN {X 0,Y 460.924,Z 639.013,A -85,B 0,C 180,E1 -8348.123,E2 -8348.123} C_VEL
LIN {X 0,Y 460.289,Z 654.967,A -85,B 0,C 180,E1 -8348.561,E2 -8348.561} C_VEL
LIN {X 0,Y 459.621,Z 669.343,A -85,B 0,C 180,E1 -8349.133,E2 -8349.133} C_VEL
LIN {X 0,Y 458.82,Z 682.918,A -85,B 0,C 180,E1 -8349.84,E2 -8349.84} C_VEL
LIN {X 0,Y 457.922,Z 696.564,A -85,B 0,C 180,E1 -8350.733,E2 -8350.733} C_VEL
LIN {X 0,Y 456.905,Z 710.421,A -85,B 0,C 180,E1 -8351.851,E2 -8351.851} C_VEL
LIN {X 0,Y 455.985,Z 722.949,A -85,B 0,C 180,E1 -8353.087,E2 -8353.087} C_VEL
LIN {X 0,Y 455.149,Z 733.448,A -85,B 0,C 180,E1 -8354.322,E2 -8354.322} C_VEL
LIN {X 0,Y 454.408,Z 743.19,A -85,B 0,C 180,E1 -8355.672,E2 -8355.672} C_VEL
LIN {X 0,Y 453.7,Z 752.753,A -85,B 0,C 180,E1 -8357.247,E2 -8357.247} C_VEL
LIN {X 0,Y 453.345,Z 760.726,A -85,B 0,C 180,E1 -8358.826,E2 -8358.826} C_VEL
LIN {X 0,Y 452.861,Z 768.16,A -85,B 0,C 180,E1 -8360.621,E2 -8360.621} C_VEL
LIN {X 0,Y 452.658,Z 774.061,A -85,B 0,C 180,E1 -8362.416,E2 -8362.416} C_VEL
LIN {X 0,Y 452.562,Z 777.566,A -85,B 0,C 180,E1 -8363.759,E2 -8363.759} C_VEL
LIN {X 0,Y 452.452,Z 781.108,A -85,B 0,C 180,E1 -8365.545,E2 -8365.545} C_VEL
LIN {X 0,Y 452.484,Z 783.44,A -85,B 0,C 180,E1 -8367.329,E2 -8367.329} C_VEL
LIN {X 0,Y 452.425,Z 784.608,A -85,B 0,C 180,E1 -8369.109,E2 -8369.109} C_VEL
LIN {X 0,Y 452.425,Z 784.601,A -85,B 0,C 180,E1 -8370.89,E2 -8370.89} C_VEL
LIN {X 0,Y 452.488,Z 783.42,A -85,B 0,C 180,E1 -8372.67,E2 -8372.67} C_VEL
LIN {X 0,Y 452.452,Z 781.078,A -85,B 0,C 180,E1 -8374.454,E2 -8374.454} C_VEL
LIN {X 0,Y 452.565,Z 777.273,A -85,B 0,C 180,E1 -8376.348,E2 -8376.348} C_VEL
LIN {X 0,Y 452.699,Z 772.687,A -85,B 0,C 180,E1 -8378.031,E2 -8378.031} C_VEL
LIN {X 0,Y 452.915,Z 766.414,A -85,B 0,C 180,E1 -8379.827,E2 -8379.827} C_VEL
LIN {X 0,Y 453.389,Z 758.542,A -85,B 0,C 180,E1 -8381.625,E2 -8381.625} C_VEL
LIN {X 0,Y 453.919,Z 750.305,A -85,B 0,C 180,E1 -8383.178,E2 -8383.178} C_VEL
LIN {X 0,Y 454.621,Z 740.085,A -85,B 0,C 180,E1 -8384.777,E2 -8384.777} C_VEL
LIN {X 0,Y 455.432,Z 729.789,A -85,B 0,C 180,E1 -8386.126,E2 -8386.126} C_VEL
LIN {X 0,Y 456.348,Z 717.938,A -85,B 0,C 180,E1 -8387.43,E2 -8387.43} C_VEL
LIN {X 0,Y 457.277,Z 705.198,A -85,B 0,C 180,E1 -8388.596,E2 -8388.596} C_VEL
LIN {X 0,Y 458.246,Z 691.794,A -85,B 0,C 180,E1 -8389.602,E2 -8389.602} C_VEL
LIN {X 0,Y 459.223,Z 676.999,A -85,B 0,C 180,E1 -8390.492,E2 -8390.492} C_VEL
LIN {X 0,Y 459.995,Z 662.179,A -85,B 0,C 180,E1 -8391.18,E2 -8391.18} C_VEL
LIN {X 0,Y 460.662,Z 647.247,A -85,B 0,C 180,E1 -8391.683,E2 -8391.683} C_VEL
LIN {X 0,Y 461.078,Z 632.335,A -85,B 0,C 180,E1 -8392.016,E2 -8392.016} C_VEL
LIN {X 0,Y 462.871,Z 498.551,A -85,B 0,C 180,E1 -8394.162,E2 -8394.162} C_VEL
LIN {X 0,Y 457.715,Z 471.853,A -85,B 0,C 180,E1 -8394.927,E2 -8394.927} C_VEL
LIN {X 0,Y 458.661,Z 456.427,A -85,B 0,C 180,E1 -8397.287,E2 -8397.287} C_VEL
LIN {X 0,Y 455.703,Z 443.332,A -85,B 0,C 180,E1 -8399.571,E2 -8399.571} C_VEL
LIN {X 0,Y 453.487,Z 434.624,A -85,B 0,C 180,E1 -8401.188,E2 -8401.188} C_VEL
LIN {X 0,Y 453.474,Z 434.624,A -85,B 0,C 180,E1 -8403.912,E2 -8403.912} C_VEL
LIN {X 0,Y 453.467,Z 434.621,A -85,B 0,C 180,E1 -8407.187,E2 -8407.187} C_VEL
LIN {X 0,Y 453.529,Z 434.614,A -85,B 0,C 180,E1 -8409.444,E2 -8409.444} C_VEL
LIN {X 0,Y 453.487,Z 434.616,A -85,B 0,C 180,E1 -8412.991,E2 -8412.991} C_VEL
LIN {X 0,Y 453.46,Z 434.626,A -85,B 0,C 180,E1 -8415.778,E2 -8415.778} C_VEL
LIN {X 0,Y 453.473,Z 434.625,A -85,B 0,C 180,E1 -8418.209,E2 -8418.209} C_VEL
LIN {X 0,Y 453.509,Z 434.619,A -85,B 0,C 180,E1 -8420.79,E2 -8420.79} C_VEL
LIN {X 0,Y 453.451,Z 434.627,A -85,B 0,C 180,E1 -8423.917,E2 -8423.917} C_VEL
LIN {X 0,Y 453.476,Z 434.618,A -85,B 0,C 180,E1 -8427.151,E2 -8427.151} C_VEL
LIN {X 0,Y 453.468,Z 434.624,A -85,B 0,C 180,E1 -8430.268,E2 -8430.268} C_VEL
LIN {X 0,Y 453.506,Z 434.613,A -85,B 0,C 180,E1 -8433.294,E2 -8433.294} C_VEL
LIN {X 0,Y 453.496,Z 434.619,A -85,B 0,C 180,E1 -8436.239,E2 -8436.239} C_VEL
LIN {X 0,Y 453.475,Z 434.617,A -85,B 0,C 180,E1 -8439.117,E2 -8439.117} C_VEL
LIN {X 0,Y 453.505,Z 434.619,A -85,B 0,C 180,E1 -8441.944,E2 -8441.944} C_VEL
LIN {X 0,Y 453.532,Z 434.616,A -85,B 0,C 180,E1 -8444.726,E2 -8444.726} C_VEL
LIN {X 0,Y 453.594,Z 434.602,A -85,B 0,C 180,E1 -8447.472,E2 -8447.472} C_VEL
LIN {X 0,Y 453.585,Z 434.605,A -85,B 0,C 180,E1 -8451.087,E2 -8451.087} C_VEL
LIN {X 0,Y 453.67,Z 434.595,A -85,B 0,C 180,E1 -8453.775,E2 -8453.775} C_VEL
LIN {X 0,Y 453.759,Z 434.581,A -85,B 0,C 180,E1 -8457.337,E2 -8457.337} C_VEL
LIN {X 0,Y 453.816,Z 434.581,A -85,B 0,C 180,E1 -8460,E2 -8460} C_VEL
LIN {X 0,Y 453.759,Z 434.589,A -85,B 0,C 180,E1 -8462.663,E2 -8462.663} C_VEL
LIN {X 0,Y 453.671,Z 434.6,A -85,B 0,C 180,E1 -8466.226,E2 -8466.226} C_VEL
LIN {X 0,Y 453.586,Z 434.608,A -85,B 0,C 180,E1 -8468.914,E2 -8468.914} C_VEL
LIN {X 0,Y 453.556,Z 434.616,A -85,B 0,C 180,E1 -8472.529,E2 -8472.529} C_VEL
LIN {X 0,Y 453.55,Z 434.616,A -85,B 0,C 180,E1 -8476.196,E2 -8476.196} C_VEL
LIN {X 0,Y 453.514,Z 434.616,A -85,B 0,C 180,E1 -8479.041,E2 -8479.041} C_VEL
LIN {X 0,Y 453.47,Z 434.622,A -85,B 0,C 180,E1 -8481.837,E2 -8481.837} C_VEL
LIN {X 0,Y 453.508,Z 434.622,A -85,B 0,C 180,E1 -8484.735,E2 -8484.735} C_VEL
LIN {X 0,Y 453.533,Z 434.617,A -85,B 0,C 180,E1 -8487.962,E2 -8487.962} C_VEL
LIN {X 0,Y 453.478,Z 434.625,A -85,B 0,C 180,E1 -8490.76,E2 -8490.76} C_VEL
LIN {X 0,Y 453.474,Z 434.624,A -85,B 0,C 180,E1 -8493.913,E2 -8493.913} C_VEL
LIN {X 0,Y 453.468,Z 434.625,A -85,B 0,C 180,E1 -8497.189,E2 -8497.189} C_VEL
LIN {X 0,Y 453.531,Z 434.625,A -85,B 0,C 180,E1 -8500.241,E2 -8500.241} C_VEL
LIN {X 0,Y 456.79,Z 448.753,A -85,B 0,C 180,E1 -8503.058,E2 -8503.058} C_VEL
LIN {X 0,Y 457.294,Z 450.393,A -85,B 0,C 180,E1 -8503.15,E2 -8503.15} C_VEL
LIN {X 0,Y 459.881,Z 456.95,A -85,B 0,C 180,E1 -8503.416,E2 -8503.416} C_VEL
LIN {X 0,Y 463.167,Z 471.345,A -85,B 0,C 180,E1 -8503.851,E2 -8503.851} C_VEL
LIN {X 0,Y 461.165,Z 613.842,A -85,B 0,C 180,E1 -8506.158,E2 -8506.158} C_VEL
LIN {X 0,Y 460.669,Z 628.928,A -85,B 0,C 180,E1 -8506.571,E2 -8506.571} C_VEL
LIN {X 0,Y 460.028,Z 643.034,A -85,B 0,C 180,E1 -8507.125,E2 -8507.125} C_VEL
LIN {X 0,Y 459.225,Z 657.846,A -85,B 0,C 180,E1 -8507.895,E2 -8507.895} C_VEL
LIN {X 0,Y 458.359,Z 670.885,A -85,B 0,C 180,E1 -8508.753,E2 -8508.753} C_VEL
LIN {X 0,Y 457.438,Z 684.025,A -85,B 0,C 180,E1 -8509.815,E2 -8509.815} C_VEL
LIN {X 0,Y 456.498,Z 696.17,A -85,B 0,C 180,E1 -8511.003,E2 -8511.003} C_VEL
LIN {X 0,Y 455.587,Z 707.415,A -85,B 0,C 180,E1 -8512.32,E2 -8512.32} C_VEL
LIN {X 0,Y 454.775,Z 717.586,A -85,B 0,C 180,E1 -8513.742,E2 -8513.742} C_VEL
LIN {X 0,Y 454.264,Z 724.419,A -85,B 0,C 180,E1 -8514.852,E2 -8514.852} C_VEL
LIN {X 0,Y 453.308,Z 727.872,A -85,B 0,C 180,E1 -8515.451,E2 -8515.451} C_VEL
LIN {X 0,Y 450.086,Z 733.253,A -85,B 0,C 180,E1 -8516.429,E2 -8516.429} C_VEL
LIN {X 0,Y 446.942,Z 738.136,A -85,B 0,C 180,E1 -8517.454,E2 -8517.454} C_VEL
LIN {X 0,Y 446.112,Z 740.819,A -85,B 0,C 180,E1 -8518.12,E2 -8518.12} C_VEL
LIN {X 0,Y 445.839,Z 746.203,A -85,B 0,C 180,E1 -8519.707,E2 -8519.707} C_VEL
LIN {X 0,Y 445.579,Z 750.437,A -85,B 0,C 180,E1 -8521.246,E2 -8521.246} C_VEL
LIN {X 0,Y 445.404,Z 753.693,A -85,B 0,C 180,E1 -8522.769,E2 -8522.769} C_VEL
LIN {X 0,Y 445.268,Z 756.681,A -85,B 0,C 180,E1 -8524.777,E2 -8524.777} C_VEL
LIN {X 0,Y 445.201,Z 758.229,A -85,B 0,C 180,E1 -8526.756,E2 -8526.756} C_VEL
LIN {X 0,Y 445.216,Z 758.422,A -85,B 0,C 180,E1 -8528.712,E2 -8528.712} C_VEL
LIN {X 0,Y 445.25,Z 757.321,A -85,B 0,C 180,E1 -8530.643,E2 -8530.643} C_VEL
LIN {X 0,Y 445.346,Z 754.949,A -85,B 0,C 180,E1 -8532.553,E2 -8532.553} C_VEL
LIN {X 0,Y 445.608,Z 751.277,A -85,B 0,C 180,E1 -8534.448,E2 -8534.448} C_VEL
LIN {X 0,Y 445.806,Z 746.292,A -85,B 0,C 180,E1 -8536.322,E2 -8536.322} C_VEL
LIN {X 0,Y 446.165,Z 739.87,A -85,B 0,C 180,E1 -8538.184,E2 -8538.184} C_VEL
LIN {X 0,Y 446.732,Z 731.83,A -85,B 0,C 180,E1 -8540.035,E2 -8540.035} C_VEL
LIN {X 0,Y 447.431,Z 722.846,A -85,B 0,C 180,E1 -8541.72,E2 -8541.72} C_VEL
LIN {X 0,Y 448.209,Z 713.046,A -85,B 0,C 180,E1 -8543.247,E2 -8543.247} C_VEL
LIN {X 0,Y 449.106,Z 702.584,A -85,B 0,C 180,E1 -8544.613,E2 -8544.613} C_VEL
LIN {X 0,Y 450.048,Z 691.242,A -85,B 0,C 180,E1 -8545.859,E2 -8545.859} C_VEL
LIN {X 0,Y 450.972,Z 679.489,A -85,B 0,C 180,E1 -8546.943,E2 -8546.943} C_VEL
LIN {X 0,Y 452.017,Z 665.544,A -85,B 0,C 180,E1 -8547.996,E2 -8547.996} C_VEL
LIN {X 0,Y 452.861,Z 651.727,A -85,B 0,C 180,E1 -8548.833,E2 -8548.833} C_VEL
LIN {X 0,Y 453.598,Z 637.557,A -85,B 0,C 180,E1 -8549.501,E2 -8549.501} C_VEL
LIN {X 0,Y 454.206,Z 622.363,A -85,B 0,C 180,E1 -8550.028,E2 -8550.028} C_VEL
LIN {X 0,Y 454.599,Z 606.37,A -85,B 0,C 180,E1 -8550.388,E2 -8550.388} C_VEL
LIN {X 0,Y 456.539,Z 471.984,A -85,B 0,C 180,E1 -8552.567,E2 -8552.567} C_VEL
LIN {X 0,Y 452.886,Z 456.974,A -85,B 0,C 180,E1 -8553.037,E2 -8553.037} C_VEL
LIN {X 0,Y 449.646,Z 448.717,A -85,B 0,C 180,E1 -8553.383,E2 -8553.383} C_VEL
LIN {X 0,Y 446.61,Z 435.478,A -85,B 0,C 180,E1 -8556.041,E2 -8556.041} C_VEL
LIN {X 0,Y 446.543,Z 435.489,A -85,B 0,C 180,E1 -8559.056,E2 -8559.056} C_VEL
LIN {X 0,Y 446.538,Z 435.487,A -85,B 0,C 180,E1 -8562.73,E2 -8562.73} C_VEL
LIN {X 0,Y 446.494,Z 435.491,A -85,B 0,C 180,E1 -8566.459,E2 -8566.459} C_VEL
LIN {X 0,Y 446.473,Z 435.496,A -85,B 0,C 180,E1 -8569.303,E2 -8569.303} C_VEL
LIN {X 0,Y 446.423,Z 435.502,A -85,B 0,C 180,E1 -8572.2,E2 -8572.2} C_VEL
LIN {X 0,Y 446.462,Z 435.492,A -85,B 0,C 180,E1 -8575.152,E2 -8575.152} C_VEL
LIN {X 0,Y 446.488,Z 435.488,A -85,B 0,C 180,E1 -8578.179,E2 -8578.179} C_VEL
LIN {X 0,Y 446.422,Z 435.503,A -85,B 0,C 180,E1 -8581.3,E2 -8581.3} C_VEL
LIN {X 0,Y 446.433,Z 435.497,A -85,B 0,C 180,E1 -8584.523,E2 -8584.523} C_VEL
LIN {X 0,Y 446.433,Z 435.493,A -85,B 0,C 180,E1 -8588.082,E2 -8588.082} C_VEL
LIN {X 0,Y 446.43,Z 435.498,A -85,B 0,C 180,E1 -8590.918,E2 -8590.918} C_VEL
LIN {X 0,Y 446.425,Z 435.5,A -85,B 0,C 180,E1 -8593.843,E2 -8593.843} C_VEL
LIN {X 0,Y 446.401,Z 435.5,A -85,B 0,C 180,E1 -8596.403,E2 -8596.403} C_VEL
LIN {X 0,Y 446.47,Z 435.497,A -85,B 0,C 180,E1 -8599.805,E2 -8599.805} C_VEL
LIN {X 0,Y 446.434,Z 435.497,A -85,B 0,C 180,E1 -8602.123,E2 -8602.123} C_VEL
LIN {X 0,Y 446.433,Z 435.497,A -85,B 0,C 180,E1 -8605.477,E2 -8605.477} C_VEL
LIN {X 0,Y 446.417,Z 435.496,A -85,B 0,C 180,E1 -8608.699,E2 -8608.699} C_VEL
LIN {X 0,Y 446.486,Z 435.494,A -85,B 0,C 180,E1 -8611.821,E2 -8611.821} C_VEL
LIN {X 0,Y 446.459,Z 435.492,A -85,B 0,C 180,E1 -8614.847,E2 -8614.847} C_VEL
LIN {X 0,Y 446.449,Z 435.494,A -85,B 0,C 180,E1 -8618.245,E2 -8618.245} C_VEL
LIN {X 0,Y 446.458,Z 435.495,A -85,B 0,C 180,E1 -8621.649,E2 -8621.649} C_VEL
LIN {X 0,Y 446.508,Z 435.482,A -85,B 0,C 180,E1 -8624.48,E2 -8624.48} C_VEL
LIN {X 0,Y 446.518,Z 435.484,A -85,B 0,C 180,E1 -8628.193,E2 -8628.193} C_VEL
LIN {X 0,Y 446.6,Z 435.478,A -85,B 0,C 180,E1 -8631.858,E2 -8631.858} C_VEL
LIN {X 0,Y 446.646,Z 435.469,A -85,B 0,C 180,E1 -8634.582,E2 -8634.582} C_VEL
LIN {X 0,Y 446.664,Z 435.467,A -85,B 0,C 180,E1 -8638.196,E2 -8638.196} C_VEL
LIN {X 0,Y 446.794,Z 435.456,A -85,B 0,C 180,E1 -8640,E2 -8640} C_VEL
LIN {X 0,Y 446.709,Z 435.458,A -85,B 0,C 180,E1 -8642.705,E2 -8642.705} C_VEL
LIN {X 0,Y 446.646,Z 435.468,A -85,B 0,C 180,E1 -8646.323,E2 -8646.323} C_VEL
LIN {X 0,Y 446.538,Z 435.484,A -85,B 0,C 180,E1 -8649.055,E2 -8649.055} C_VEL
LIN {X 0,Y 446.521,Z 435.477,A -85,B 0,C 180,E1 -8652.73,E2 -8652.73} C_VEL
LIN {X 0,Y 446.496,Z 435.489,A -85,B 0,C 180,E1 -8656.228,E2 -8656.228} C_VEL
LIN {X 0,Y 446.469,Z 435.485,A -85,B 0,C 180,E1 -8659.303,E2 -8659.303} C_VEL
LIN {X 0,Y 446.417,Z 435.499,A -85,B 0,C 180,E1 -8662.199,E2 -8662.199} C_VEL
LIN {X 0,Y 446.457,Z 435.495,A -85,B 0,C 180,E1 -8665.152,E2 -8665.152} C_VEL
LIN {X 0,Y 446.484,Z 435.491,A -85,B 0,C 180,E1 -8668.178,E2 -8668.178} C_VEL
LIN {X 0,Y 446.417,Z 435.5,A -85,B 0,C 180,E1 -8671.3,E2 -8671.3} C_VEL
LIN {X 0,Y 446.43,Z 435.498,A -85,B 0,C 180,E1 -8674.523,E2 -8674.523} C_VEL
LIN {X 0,Y 446.43,Z 435.501,A -85,B 0,C 180,E1 -8678.082,E2 -8678.082} C_VEL
LIN {X 0,Y 446.426,Z 435.498,A -85,B 0,C 180,E1 -8680.917,E2 -8680.917} C_VEL
LIN {X 0,Y 446.401,Z 435.506,A -85,B 0,C 180,E1 -8683.846,E2 -8683.846} C_VEL
LIN {X 0,Y 446.447,Z 435.497,A -85,B 0,C 180,E1 -8686.397,E2 -8686.397} C_VEL
LIN {X 0,Y 446.443,Z 435.501,A -85,B 0,C 180,E1 -8689.802,E2 -8689.802} C_VEL
LIN {X 0,Y 446.402,Z 435.501,A -85,B 0,C 180,E1 -8693.255,E2 -8693.255} C_VEL
LIN {X 0,Y 446.448,Z 435.502,A -85,B 0,C 180,E1 -8696.566,E2 -8696.566} C_VEL
LIN {X 0,Y 446.468,Z 435.631,A -85,B 0,C 180,E1 -8698.529,E2 -8698.529} C_VEL
LIN {X 0,Y 450.413,Z 451.514,A -85,B 0,C 180,E1 -8701.414,E2 -8701.414} C_VEL
LIN {X 0,Y 451.845,Z 458.714,A -85,B 0,C 180,E1 -8702.66,E2 -8702.66} C_VEL
LIN {X 0,Y 450.949,Z 472.136,A -85,B 0,C 180,E1 -8704.733,E2 -8704.733} C_VEL
LIN {X 0,Y 456.28,Z 500.108,A -85,B 0,C 180,E1 -8705.522,E2 -8705.522} C_VEL
LIN {X 0,Y 454.336,Z 638.536,A -85,B 0,C 180,E1 -8707.789,E2 -8707.789} C_VEL
LIN {X 0,Y 453.653,Z 654.666,A -85,B 0,C 180,E1 -8708.235,E2 -8708.235} C_VEL
LIN {X 0,Y 452.948,Z 669.585,A -85,B 0,C 180,E1 -8708.84,E2 -8708.84} C_VEL
LIN {X 0,Y 452,Z 684.499,A -85,B 0,C 180,E1 -8709.641,E2 -8709.641} C_VEL
LIN {X 0,Y 451.069,Z 697.84,A -85,B 0,C 180,E1 -8710.546,E2 -8710.546} C_VEL
LIN {X 0,Y 449.997,Z 711.404,A -85,B 0,C 180,E1 -8711.681,E2 -8711.681} C_VEL
LIN {X 0,Y 449.045,Z 723.767,A -85,B 0,C 180,E1 -8712.938,E2 -8712.938} C_VEL
LIN {X 0,Y 448.092,Z 734.992,A -85,B 0,C 180,E1 -8714.302,E2 -8714.302} C_VEL
LIN {X 0,Y 447.238,Z 745.919,A -85,B 0,C 180,E1 -8715.902,E2 -8715.902} C_VEL
LIN {X 0,Y 446.512,Z 755.273,A -85,B 0,C 180,E1 -8717.555,E2 -8717.555} C_VEL
LIN {X 0,Y 446.142,Z 762.539,A -85,B 0,C 180,E1 -8719.103,E2 -8719.103} C_VEL
LIN {X 0,Y 445.729,Z 769.571,A -85,B 0,C 180,E1 -8720.928,E2 -8720.928} C_VEL
LIN {X 0,Y 445.571,Z 775.104,A -85,B 0,C 180,E1 -8722.75,E2 -8722.75} C_VEL
LIN {X 0,Y 445.419,Z 779.283,A -85,B 0,C 180,E1 -8724.567,E2 -8724.567} C_VEL
LIN {X 0,Y 445.337,Z 782.212,A -85,B 0,C 180,E1 -8726.38,E2 -8726.38} C_VEL
LIN {X 0,Y 445.348,Z 783.959,A -85,B 0,C 180,E1 -8728.191,E2 -8728.191} C_VEL
LIN {X 0,Y 445.339,Z 784.553,A -85,B 0,C 180,E1 -8730,E2 -8730} C_VEL
LIN {X 0,Y 445.348,Z 783.945,A -85,B 0,C 180,E1 -8731.808,E2 -8731.808} C_VEL
LIN {X 0,Y 445.359,Z 782.187,A -85,B 0,C 180,E1 -8733.618,E2 -8733.618} C_VEL
LIN {X 0,Y 445.419,Z 779.251,A -85,B 0,C 180,E1 -8735.432,E2 -8735.432} C_VEL
LIN {X 0,Y 445.57,Z 775.068,A -85,B 0,C 180,E1 -8737.249,E2 -8737.249} C_VEL
LIN {X 0,Y 445.727,Z 769.525,A -85,B 0,C 180,E1 -8739.071,E2 -8739.071} C_VEL
LIN {X 0,Y 446.139,Z 762.478,A -85,B 0,C 180,E1 -8740.896,E2 -8740.896} C_VEL
LIN {X 0,Y 446.548,Z 754.215,A -85,B 0,C 180,E1 -8742.635,E2 -8742.635} C_VEL
LIN {X 0,Y 447.228,Z 745.864,A -85,B 0,C 180,E1 -8744.097,E2 -8744.097} C_VEL
LIN {X 0,Y 448.056,Z 734.953,A -85,B 0,C 180,E1 -8745.698,E2 -8745.698} C_VEL
LIN {X 0,Y 449.067,Z 723.728,A -85,B 0,C 180,E1 -8747.063,E2 -8747.063} C_VEL
LIN {X 0,Y 449.98,Z 711.426,A -85,B 0,C 180,E1 -8748.319,E2 -8748.319} C_VEL
LIN {X 0,Y 451.063,Z 697.905,A -85,B 0,C 180,E1 -8749.453,E2 -8749.453} C_VEL
LIN {X 0,Y 452.037,Z 684.625,A -85,B 0,C 180,E1 -8750.357,E2 -8750.357} C_VEL
LIN {X 0,Y 452.962,Z 669.821,A -85,B 0,C 180,E1 -8751.159,E2 -8751.159} C_VEL
LIN {X 0,Y 453.725,Z 654.488,A -85,B 0,C 180,E1 -8751.785,E2 -8751.785} C_VEL
LIN {X 0,Y 454.323,Z 639.353,A -85,B 0,C 180,E1 -8752.211,E2 -8752.211} C_VEL
LIN {X 0,Y 455.157,Z 589.93,A -85,B 0,C 180,E1 -8753.036,E2 -8753.036} C_VEL
LIN {X 0,Y 456.274,Z 498.815,A -85,B 0,C 180,E1 -8754.531,E2 -8754.531} C_VEL
LIN {X 0,Y 450.935,Z 471.75,A -85,B 0,C 180,E1 -8755.318,E2 -8755.318} C_VEL
LIN {X 0,Y 451.866,Z 458.696,A -85,B 0,C 180,E1 -8757.339,E2 -8757.339} C_VEL
LIN {X 0,Y 449.593,Z 447.887,A -85,B 0,C 180,E1 -8759.24,E2 -8759.24} C_VEL
LIN {X 0,Y 446.439,Z 435.5,A -85,B 0,C 180,E1 -8761.56,E2 -8761.56} C_VEL
LIN {X 0,Y 446.427,Z 435.504,A -85,B 0,C 180,E1 -8764.522,E2 -8764.522} C_VEL
LIN {X 0,Y 446.434,Z 435.499,A -85,B 0,C 180,E1 -8768.083,E2 -8768.083} C_VEL
LIN {X 0,Y 446.443,Z 435.5,A -85,B 0,C 180,E1 -8770.92,E2 -8770.92} C_VEL
LIN {X 0,Y 446.44,Z 435.496,A -85,B 0,C 180,E1 -8773.84,E2 -8773.84} C_VEL
LIN {X 0,Y 446.393,Z 435.5,A -85,B 0,C 180,E1 -8776.403,E2 -8776.403} C_VEL
LIN {X 0,Y 446.421,Z 435.5,A -85,B 0,C 180,E1 -8779.082,E2 -8779.082} C_VEL
LIN {X 0,Y 446.424,Z 435.502,A -85,B 0,C 180,E1 -8781.918,E2 -8781.918} C_VEL
LIN {X 0,Y 446.424,Z 435.499,A -85,B 0,C 180,E1 -8785.477,E2 -8785.477} C_VEL
LIN {X 0,Y 446.409,Z 435.503,A -85,B 0,C 180,E1 -8788.699,E2 -8788.699} C_VEL
LIN {X 0,Y 446.477,Z 435.494,A -85,B 0,C 180,E1 -8791.821,E2 -8791.821} C_VEL
LIN {X 0,Y 446.451,Z 435.496,A -85,B 0,C 180,E1 -8794.848,E2 -8794.848} C_VEL
LIN {X 0,Y 446.441,Z 435.503,A -85,B 0,C 180,E1 -8798.245,E2 -8798.245} C_VEL
LIN {X 0,Y 446.45,Z 435.496,A -85,B 0,C 180,E1 -8801.649,E2 -8801.649} C_VEL
LIN {X 0,Y 446.5,Z 435.495,A -85,B 0,C 180,E1 -8804.48,E2 -8804.48} C_VEL
LIN {X 0,Y 446.532,Z 435.488,A -85,B 0,C 180,E1 -8808.194,E2 -8808.194} C_VEL
LIN {X 0,Y 446.593,Z 435.478,A -85,B 0,C 180,E1 -8811.858,E2 -8811.858} C_VEL
LIN {X 0,Y 446.639,Z 435.474,A -85,B 0,C 180,E1 -8814.583,E2 -8814.583} C_VEL
LIN {X 0,Y 446.703,Z 435.46,A -85,B 0,C 180,E1 -8817.295,E2 -8817.295} C_VEL
LIN {X 0,Y 446.786,Z 435.456,A -85,B 0,C 180,E1 -8820,E2 -8820} C_VEL
LIN {X 0,Y 446.703,Z 435.467,A -85,B 0,C 180,E1 -8822.706,E2 -8822.706} C_VEL
LIN {X 0,Y 446.64,Z 435.477,A -85,B 0,C 180,E1 -8826.324,E2 -8826.324} C_VEL
LIN {X 0,Y 446.531,Z 435.486,A -85,B 0,C 180,E1 -8829.056,E2 -8829.056} C_VEL
LIN {X 0,Y 446.515,Z 435.49,A -85,B 0,C 180,E1 -8832.73,E2 -8832.73} C_VEL
LIN {X 0,Y 446.512,Z 435.492,A -85,B 0,C 180,E1 -8836.239,E2 -8836.239} C_VEL
LIN {X 0,Y 446.463,Z 435.493,A -85,B 0,C 180,E1 -8839.304,E2 -8839.304} C_VEL
LIN {X 0,Y 446.412,Z 435.504,A -85,B 0,C 180,E1 -8842.2,E2 -8842.2} C_VEL
LIN {X 0,Y 446.452,Z 435.498,A -85,B 0,C 180,E1 -8845.153,E2 -8845.153} C_VEL
LIN {X 0,Y 446.479,Z 435.498,A -85,B 0,C 180,E1 -8848.179,E2 -8848.179} C_VEL
LIN {X 0,Y 446.415,Z 435.502,A -85,B 0,C 180,E1 -8851.301,E2 -8851.301} C_VEL
LIN {X 0,Y 446.426,Z 435.501,A -85,B 0,C 180,E1 -8854.524,E2 -8854.524} C_VEL
LIN {X 0,Y 446.435,Z 435.505,A -85,B 0,C 180,E1 -8858.084,E2 -8858.084} C_VEL
LIN {X 0,Y 446.545,Z 435.655,A -85,B 0,C 180,E1 -8859.91,E2 -8859.91} C_VEL
LIN {X 0,Y 449.729,Z 449.377,A -85,B 0,C 180,E1 -8862.67,E2 -8862.67} C_VEL
LIN {X 0,Y 453.757,Z 459.532,A -85,B 0,C 180,E1 -8863.096,E2 -8863.096} C_VEL
LIN {X 0,Y 456.737,Z 472.997,A -85,B 0,C 180,E1 -8863.507,E2 -8863.507} C_VEL
LIN {X 0,Y 454.581,Z 614.437,A -85,B 0,C 180,E1 -8865.832,E2 -8865.832} C_VEL
LIN {X 0,Y 454.032,Z 629.897,A -85,B 0,C 180,E1 -8866.267,E2 -8866.267} C_VEL
LIN {X 0,Y 453.346,Z 644.796,A -85,B 0,C 180,E1 -8866.874,E2 -8866.874} C_VEL
LIN {X 0,Y 452.49,Z 659.161,A -85,B 0,C 180,E1 -8867.649,E2 -8867.649} C_VEL
LIN {X 0,Y 451.518,Z 673.204,A -85,B 0,C 180,E1 -8868.609,E2 -8868.609} C_VEL
LIN {X 0,Y 450.478,Z 686.781,A -85,B 0,C 180,E1 -8869.761,E2 -8869.761} C_VEL
LIN {X 0,Y 449.506,Z 698.834,A -85,B 0,C 180,E1 -8871.002,E2 -8871.002} C_VEL
LIN {X 0,Y 448.574,Z 709.682,A -85,B 0,C 180,E1 -8872.337,E2 -8872.337} C_VEL
LIN {X 0,Y 447.796,Z 718.791,A -85,B 0,C 180,E1 -8873.668,E2 -8873.668} C_VEL
LIN {X 0,Y 447.04,Z 727.461,A -85,B 0,C 180,E1 -8875.159,E2 -8875.159} C_VEL
LIN {X 0,Y 446.514,Z 735.6,A -85,B 0,C 180,E1 -8876.843,E2 -8876.843} C_VEL
LIN {X 0,Y 446.112,Z 740.819,A -85,B 0,C 180,E1 -8878.12,E2 -8878.12} C_VEL
LIN {X 0,Y 445.294,Z 743.356,A -85,B 0,C 180,E1 -8878.799,E2 -8878.799} C_VEL
LIN {X 0,Y 440.867,Z 748.541,A -85,B 0,C 180,E1 -8880.368,E2 -8880.368} C_VEL
LIN {X 0,Y 438.791,Z 751.038,A -85,B 0,C 180,E1 -8881.311,E2 -8881.311} C_VEL
LIN {X 0,Y 438.411,Z 752.176,A -85,B 0,C 180,E1 -8881.802,E2 -8881.802} C_VEL
LIN {X 0,Y 438.208,Z 755.907,A -85,B 0,C 180,E1 -8883.914,E2 -8883.914} C_VEL
LIN {X 0,Y 438.12,Z 758.119,A -85,B 0,C 180,E1 -8886.115,E2 -8886.115} C_VEL
LIN {X 0,Y 438.097,Z 758.636,A -85,B 0,C 180,E1 -8887.356,E2 -8887.356} C_VEL
LIN {X 0,Y 438.113,Z 758.431,A -85,B 0,C 180,E1 -8889.335,E2 -8889.335} C_VEL
LIN {X 0,Y 438.222,Z 756.94,A -85,B 0,C 180,E1 -8891.292,E2 -8891.292} C_VEL
LIN {X 0,Y 438.322,Z 754.183,A -85,B 0,C 180,E1 -8893.226,E2 -8893.226} C_VEL
LIN {X 0,Y 438.588,Z 750.106,A -85,B 0,C 180,E1 -8895.145,E2 -8895.145} C_VEL
LIN {X 0,Y 438.836,Z 744.684,A -85,B 0,C 180,E1 -8897.044,E2 -8897.044} C_VEL
LIN {X 0,Y 439.314,Z 737.776,A -85,B 0,C 180,E1 -8898.933,E2 -8898.933} C_VEL
LIN {X 0,Y 439.854,Z 730.35,A -85,B 0,C 180,E1 -8900.575,E2 -8900.575} C_VEL
LIN {X 0,Y 440.63,Z 721.318,A -85,B 0,C 180,E1 -8902.231,E2 -8902.231} C_VEL
LIN {X 0,Y 441.543,Z 710.8,A -85,B 0,C 180,E1 -8903.833,E2 -8903.833} C_VEL
LIN {X 0,Y 442.545,Z 699.848,A -85,B 0,C 180,E1 -8905.218,E2 -8905.218} C_VEL
LIN {X 0,Y 443.397,Z 689.122,A -85,B 0,C 180,E1 -8906.365,E2 -8906.365} C_VEL
LIN {X 0,Y 444.483,Z 676.319,A -85,B 0,C 180,E1 -8907.508,E2 -8907.508} C_VEL
LIN {X 0,Y 445.534,Z 662.239,A -85,B 0,C 180,E1 -8908.532,E2 -8908.532} C_VEL
LIN {X 0,Y 446.485,Z 647.428,A -85,B 0,C 180,E1 -8909.38,E2 -8909.38} C_VEL
LIN {X 0,Y 447.246,Z 632.533,A -85,B 0,C 180,E1 -8910.029,E2 -8910.029} C_VEL
LIN {X 0,Y 447.787,Z 618.116,A -85,B 0,C 180,E1 -8910.478,E2 -8910.478} C_VEL
LIN {X 0,Y 448.131,Z 599.533,A -85,B 0,C 180,E1 -8910.843,E2 -8910.843} C_VEL
LIN {X 0,Y 450.021,Z 473.121,A -85,B 0,C 180,E1 -8912.924,E2 -8912.924} C_VEL
LIN {X 0,Y 446.827,Z 459.742,A -85,B 0,C 180,E1 -8913.348,E2 -8913.348} C_VEL
LIN {X 0,Y 442.423,Z 448.913,A -85,B 0,C 180,E1 -8913.823,E2 -8913.823} C_VEL
LIN {X 0,Y 439.574,Z 436.358,A -85,B 0,C 180,E1 -8916.397,E2 -8916.397} C_VEL
LIN {X 0,Y 439.505,Z 436.367,A -85,B 0,C 180,E1 -8919.202,E2 -8919.202} C_VEL
LIN {X 0,Y 439.508,Z 436.363,A -85,B 0,C 180,E1 -8922.727,E2 -8922.727} C_VEL
LIN {X 0,Y 439.451,Z 436.369,A -85,B 0,C 180,E1 -8926.349,E2 -8926.349} C_VEL
LIN {X 0,Y 439.435,Z 436.377,A -85,B 0,C 180,E1 -8929.625,E2 -8929.625} C_VEL
LIN {X 0,Y 439.37,Z 436.379,A -85,B 0,C 180,E1 -8932.575,E2 -8932.575} C_VEL
LIN {X 0,Y 439.41,Z 436.375,A -85,B 0,C 180,E1 -8935.585,E2 -8935.585} C_VEL
LIN {X 0,Y 439.425,Z 436.366,A -85,B 0,C 180,E1 -8938.673,E2 -8938.673} C_VEL
LIN {X 0,Y 439.377,Z 436.373,A -85,B 0,C 180,E1 -8941.86,E2 -8941.86} C_VEL
LIN {X 0,Y 439.404,Z 436.375,A -85,B 0,C 180,E1 -8945.156,E2 -8945.156} C_VEL
LIN {X 0,Y 439.393,Z 436.367,A -85,B 0,C 180,E1 -8948.594,E2 -8948.594} C_VEL
LIN {X 0,Y 439.392,Z 436.377,A -85,B 0,C 180,E1 -8951.257,E2 -8951.257} C_VEL
LIN {X 0,Y 439.408,Z 436.371,A -85,B 0,C 180,E1 -8954.728,E2 -8954.728} C_VEL
LIN {X 0,Y 439.399,Z 436.371,A -85,B 0,C 180,E1 -8957.796,E2 -8957.796} C_VEL
LIN {X 0,Y 439.451,Z 436.368,A -85,B 0,C 180,E1 -8960.23,E2 -8960.23} C_VEL
LIN {X 0,Y 439.379,Z 436.373,A -85,B 0,C 180,E1 -8963.713,E2 -8963.713} C_VEL
LIN {X 0,Y 439.374,Z 436.377,A -85,B 0,C 180,E1 -8967.054,E2 -8967.054} C_VEL
LIN {X 0,Y 439.383,Z 436.369,A -85,B 0,C 180,E1 -8970.274,E2 -8970.274} C_VEL
LIN {X 0,Y 439.431,Z 436.373,A -85,B 0,C 180,E1 -8973.396,E2 -8973.396} C_VEL
LIN {X 0,Y 439.387,Z 436.364,A -85,B 0,C 180,E1 -8976.429,E2 -8976.429} C_VEL
LIN {X 0,Y 439.389,Z 436.376,A -85,B 0,C 180,E1 -8979.397,E2 -8979.397} C_VEL
LIN {X 0,Y 439.432,Z 436.363,A -85,B 0,C 180,E1 -8982.309,E2 -8982.309} C_VEL
LIN {X 0,Y 439.448,Z 436.363,A -85,B 0,C 180,E1 -8985.174,E2 -8985.174} C_VEL
LIN {X 0,Y 439.484,Z 436.362,A -85,B 0,C 180,E1 -8988.001,E2 -8988.001} C_VEL
LIN {X 0,Y 439.548,Z 436.354,A -85,B 0,C 180,E1 -8991.726,E2 -8991.726} C_VEL
LIN {X 0,Y 439.621,Z 436.344,A -85,B 0,C 180,E1 -8994.496,E2 -8994.496} C_VEL
LIN {X 0,Y 439.634,Z 436.342,A -85,B 0,C 180,E1 -8998.168,E2 -8998.168} C_VEL
LIN {X 0,Y 439.764,Z 436.331,A -85,B 0,C 180,E1 -9000,E2 -9000} C_VEL
LIN {X 0,Y 439.656,Z 436.336,A -85,B 0,C 180,E1 -9002.748,E2 -9002.748} C_VEL
LIN {X 0,Y 439.617,Z 436.343,A -85,B 0,C 180,E1 -9006.425,E2 -9006.425} C_VEL
LIN {X 0,Y 439.499,Z 436.362,A -85,B 0,C 180,E1 -9009.201,E2 -9009.201} C_VEL
LIN {X 0,Y 439.465,Z 436.357,A -85,B 0,C 180,E1 -9012.937,E2 -9012.937} C_VEL
LIN {X 0,Y 439.447,Z 436.366,A -85,B 0,C 180,E1 -9016.349,E2 -9016.349} C_VEL
LIN {X 0,Y 439.402,Z 436.369,A -85,B 0,C 180,E1 -9019.626,E2 -9019.626} C_VEL
LIN {X 0,Y 439.364,Z 436.376,A -85,B 0,C 180,E1 -9022.575,E2 -9022.575} C_VEL
LIN {X 0,Y 439.405,Z 436.377,A -85,B 0,C 180,E1 -9025.585,E2 -9025.585} C_VEL
LIN {X 0,Y 439.421,Z 436.369,A -85,B 0,C 180,E1 -9028.673,E2 -9028.673} C_VEL
LIN {X 0,Y 439.372,Z 436.382,A -85,B 0,C 180,E1 -9031.86,E2 -9031.86} C_VEL
LIN {X 0,Y 439.401,Z 436.375,A -85,B 0,C 180,E1 -9035.156,E2 -9035.156} C_VEL
LIN {X 0,Y 439.39,Z 436.374,A -85,B 0,C 180,E1 -9038.594,E2 -9038.594} C_VEL
LIN {X 0,Y 439.388,Z 436.377,A -85,B 0,C 180,E1 -9041.257,E2 -9041.257} C_VEL
LIN {X 0,Y 439.402,Z 436.373,A -85,B 0,C 180,E1 -9044.729,E2 -9044.729} C_VEL
LIN {X 0,Y 439.411,Z 436.376,A -85,B 0,C 180,E1 -9047.797,E2 -9047.797} C_VEL
LIN {X 0,Y 439.426,Z 436.374,A -85,B 0,C 180,E1 -9050.227,E2 -9050.227} C_VEL
LIN {X 0,Y 439.373,Z 436.378,A -85,B 0,C 180,E1 -9053.713,E2 -9053.713} C_VEL
LIN {X 0,Y 439.373,Z 436.384,A -85,B 0,C 180,E1 -9057.054,E2 -9057.054} C_VEL
LIN {X 0,Y 439.391,Z 436.401,A -85,B 0,C 180,E1 -9058.141,E2 -9058.141} C_VEL
LIN {X 0,Y 443.228,Z 451.711,A -85,B 0,C 180,E1 -9060.983,E2 -9060.983} C_VEL
LIN {X 0,Y 444.979,Z 459.855,A -85,B 0,C 180,E1 -9062.428,E2 -9062.428} C_VEL
LIN {X 0,Y 444.221,Z 471.937,A -85,B 0,C 180,E1 -9064.329,E2 -9064.329} C_VEL
LIN {X 0,Y 449.764,Z 500.522,A -85,B 0,C 180,E1 -9065.16,E2 -9065.16} C_VEL
LIN {X 0,Y 447.954,Z 626.951,A -85,B 0,C 180,E1 -9067.242,E2 -9067.242} C_VEL
LIN {X 0,Y 447.535,Z 643.809,A -85,B 0,C 180,E1 -9067.585,E2 -9067.585} C_VEL
LIN {X 0,Y 446.857,Z 658.831,A -85,B 0,C 180,E1 -9068.067,E2 -9068.067} C_VEL
LIN {X 0,Y 445.998,Z 674.047,A -85,B 0,C 180,E1 -9068.75,E2 -9068.75} C_VEL
LIN {X 0,Y 445.048,Z 687.742,A -85,B 0,C 180,E1 -9069.55,E2 -9069.55} C_VEL
LIN {X 0,Y 443.976,Z 701.859,A -85,B 0,C 180,E1 -9070.584,E2 -9070.584} C_VEL
LIN {X 0,Y 442.887,Z 714.675,A -85,B 0,C 180,E1 -9071.735,E2 -9071.735} C_VEL
LIN {X 0,Y 441.989,Z 725.908,A -85,B 0,C 180,E1 -9072.948,E2 -9072.948} C_VEL
LIN {X 0,Y 441.005,Z 736.392,A -85,B 0,C 180,E1 -9074.281,E2 -9074.281} C_VEL
LIN {X 0,Y 440.147,Z 747.042,A -85,B 0,C 180,E1 -9075.906,E2 -9075.906} C_VEL
LIN {X 0,Y 439.437,Z 756.426,A -85,B 0,C 180,E1 -9077.639,E2 -9077.639} C_VEL
LIN {X 0,Y 439.126,Z 762.313,A -85,B 0,C 180,E1 -9078.927,E2 -9078.927} C_VEL
LIN {X 0,Y 438.663,Z 769.352,A -85,B 0,C 180,E1 -9080.78,E2 -9080.78} C_VEL
LIN {X 0,Y 438.487,Z 774.89,A -85,B 0,C 180,E1 -9082.633,E2 -9082.633} C_VEL
LIN {X 0,Y 438.322,Z 779.073,A -85,B 0,C 180,E1 -9084.479,E2 -9084.479} C_VEL
LIN {X 0,Y 438.24,Z 782.004,A -85,B 0,C 180,E1 -9086.322,E2 -9086.322} C_VEL
LIN {X 0,Y 438.27,Z 783.752,A -85,B 0,C 180,E1 -9088.162,E2 -9088.162} C_VEL
LIN {X 0,Y 438.25,Z 784.346,A -85,B 0,C 180,E1 -9089.999,E2 -9089.999} C_VEL
LIN {X 0,Y 438.271,Z 783.738,A -85,B 0,C 180,E1 -9091.837,E2 -9091.837} C_VEL
LIN {X 0,Y 438.26,Z 781.978,A -85,B 0,C 180,E1 -9093.677,E2 -9093.677} C_VEL
LIN {X 0,Y 438.325,Z 779.042,A -85,B 0,C 180,E1 -9095.52,E2 -9095.52} C_VEL
LIN {X 0,Y 438.486,Z 774.86,A -85,B 0,C 180,E1 -9097.366,E2 -9097.366} C_VEL
LIN {X 0,Y 438.662,Z 769.318,A -85,B 0,C 180,E1 -9099.219,E2 -9099.219} C_VEL
LIN {X 0,Y 439.122,Z 762.274,A -85,B 0,C 180,E1 -9101.072,E2 -9101.072} C_VEL
LIN {X 0,Y 439.65,Z 753.509,A -85,B 0,C 180,E1 -9102.931,E2 -9102.931} C_VEL
LIN {X 0,Y 440.385,Z 744.204,A -85,B 0,C 180,E1 -9104.557,E2 -9104.557} C_VEL
LIN {X 0,Y 441.155,Z 734.748,A -85,B 0,C 180,E1 -9105.95,E2 -9105.95} C_VEL
LIN {X 0,Y 442.234,Z 723.051,A -85,B 0,C 180,E1 -9107.391,E2 -9107.391} C_VEL
LIN {X 0,Y 443.268,Z 709.985,A -85,B 0,C 180,E1 -9108.726,E2 -9108.726} C_VEL
LIN {X 0,Y 444.316,Z 697.703,A -85,B 0,C 180,E1 -9109.76,E2 -9109.76} C_VEL
LIN {X 0,Y 445.338,Z 684.433,A -85,B 0,C 180,E1 -9110.677,E2 -9110.677} C_VEL
LIN {X 0,Y 446.306,Z 670.135,A -85,B 0,C 180,E1 -9111.465,E2 -9111.465} C_VEL
LIN {X 0,Y 447.087,Z 655.149,A -85,B 0,C 180,E1 -9112.094,E2 -9112.094} C_VEL
LIN {X 0,Y 447.712,Z 640.414,A -85,B 0,C 180,E1 -9112.526,E2 -9112.526} C_VEL
LIN {X 0,Y 448.183,Z 616.549,A -85,B 0,C 180,E1 -9112.958,E2 -9112.958} C_VEL
LIN {X 0,Y 449.959,Z 501.25,A -85,B 0,C 180,E1 -9114.858,E2 -9114.858} C_VEL
LIN {X 0,Y 444.811,Z 474.33,A -85,B 0,C 180,E1 -9115.649,E2 -9115.649} C_VEL
LIN {X 0,Y 444.222,Z 471.449,A -85,B 0,C 180,E1 -9115.748,E2 -9115.748} C_VEL
LIN {X 0,Y 444.999,Z 459.872,A -85,B 0,C 180,E1 -9117.577,E2 -9117.577} C_VEL
LIN {X 0,Y 442.309,Z 447.738,A -85,B 0,C 180,E1 -9119.77,E2 -9119.77} C_VEL
LIN {X 0,Y 439.375,Z 436.38,A -85,B 0,C 180,E1 -9121.948,E2 -9121.948} C_VEL
LIN {X 0,Y 439.397,Z 436.374,A -85,B 0,C 180,E1 -9125.155,E2 -9125.155} C_VEL
LIN {X 0,Y 439.395,Z 436.379,A -85,B 0,C 180,E1 -9128.592,E2 -9128.592} C_VEL
LIN {X 0,Y 439.4,Z 436.376,A -85,B 0,C 180,E1 -9131.259,E2 -9131.259} C_VEL
LIN {X 0,Y 439.403,Z 436.378,A -85,B 0,C 180,E1 -9134.728,E2 -9134.728} C_VEL
LIN {X 0,Y 439.39,Z 436.374,A -85,B 0,C 180,E1 -9137.795,E2 -9137.795} C_VEL
LIN {X 0,Y 439.43,Z 436.374,A -85,B 0,C 180,E1 -9140.228,E2 -9140.228} C_VEL
LIN {X 0,Y 439.371,Z 436.379,A -85,B 0,C 180,E1 -9143.713,E2 -9143.713} C_VEL
LIN {X 0,Y 439.365,Z 436.376,A -85,B 0,C 180,E1 -9147.054,E2 -9147.054} C_VEL
LIN {X 0,Y 439.375,Z 436.379,A -85,B 0,C 180,E1 -9150.274,E2 -9150.274} C_VEL
LIN {X 0,Y 439.423,Z 436.368,A -85,B 0,C 180,E1 -9153.396,E2 -9153.396} C_VEL
LIN {X 0,Y 439.38,Z 436.378,A -85,B 0,C 180,E1 -9156.429,E2 -9156.429} C_VEL
LIN {X 0,Y 439.381,Z 436.372,A -85,B 0,C 180,E1 -9159.397,E2 -9159.397} C_VEL
LIN {X 0,Y 439.424,Z 436.373,A -85,B 0,C 180,E1 -9162.309,E2 -9162.309} C_VEL
LIN {X 0,Y 439.44,Z 436.368,A -85,B 0,C 180,E1 -9165.174,E2 -9165.174} C_VEL
LIN {X 0,Y 439.5,Z 436.362,A -85,B 0,C 180,E1 -9168.002,E2 -9168.002} C_VEL
LIN {X 0,Y 439.54,Z 436.355,A -85,B 0,C 180,E1 -9171.726,E2 -9171.726} C_VEL
LIN {X 0,Y 439.614,Z 436.348,A -85,B 0,C 180,E1 -9174.496,E2 -9174.496} C_VEL
LIN {X 0,Y 439.629,Z 436.345,A -85,B 0,C 180,E1 -9178.168,E2 -9178.168} C_VEL
LIN {X 0,Y 439.756,Z 436.332,A -85,B 0,C 180,E1 -9180,E2 -9180} C_VEL
LIN {X 0,Y 439.65,Z 436.346,A -85,B 0,C 180,E1 -9182.749,E2 -9182.749} C_VEL
LIN {X 0,Y 439.612,Z 436.353,A -85,B 0,C 180,E1 -9186.426,E2 -9186.426} C_VEL
LIN {X 0,Y 439.493,Z 436.362,A -85,B 0,C 180,E1 -9189.202,E2 -9189.202} C_VEL
LIN {X 0,Y 439.459,Z 436.367,A -85,B 0,C 180,E1 -9192.938,E2 -9192.938} C_VEL
LIN {X 0,Y 439.454,Z 436.37,A -85,B 0,C 180,E1 -9196.355,E2 -9196.355} C_VEL
LIN {X 0,Y 439.396,Z 436.374,A -85,B 0,C 180,E1 -9199.627,E2 -9199.627} C_VEL
LIN {X 0,Y 439.359,Z 436.386,A -85,B 0,C 180,E1 -9202.576,E2 -9202.576} C_VEL
LIN {X 0,Y 439.4,Z 436.376,A -85,B 0,C 180,E1 -9205.586,E2 -9205.586} C_VEL
LIN {X 0,Y 439.42,Z 436.376,A -85,B 0,C 180,E1 -9208.674,E2 -9208.674} C_VEL
LIN {X 0,Y 439.378,Z 436.38,A -85,B 0,C 180,E1 -9212.034,E2 -9212.034} C_VEL
LIN {X 0,Y 439.392,Z 436.378,A -85,B 0,C 180,E1 -9215.342,E2 -9215.342} C_VEL
LIN {X 0,Y 439.434,Z 436.375,A -85,B 0,C 180,E1 -9219.179,E2 -9219.179} C_VEL
LIN {X 0,Y 439.46,Z 436.465,A -85,B 0,C 180,E1 -9219.509,E2 -9219.509} C_VEL
LIN {X 0,Y 442.564,Z 449.495,A -85,B 0,C 180,E1 -9222.217,E2 -9222.217} C_VEL
LIN {X 0,Y 447.637,Z 462.045,A -85,B 0,C 180,E1 -9222.764,E2 -9222.764} C_VEL
LIN {X 0,Y 450.227,Z 473.438,A -85,B 0,C 180,E1 -9223.126,E2 -9223.126} C_VEL
LIN {X 0,Y 448.055,Z 614.348,A -85,B 0,C 180,E1 -9225.478,E2 -9225.478} C_VEL
LIN {X 0,Y 447.526,Z 629.406,A -85,B 0,C 180,E1 -9225.903,E2 -9225.903} C_VEL
LIN {X 0,Y 446.838,Z 643.057,A -85,B 0,C 180,E1 -9226.453,E2 -9226.453} C_VEL
LIN {X 0,Y 446.017,Z 657.085,A -85,B 0,C 180,E1 -9227.194,E2 -9227.194} C_VEL
LIN {X 0,Y 445.085,Z 669.99,A -85,B 0,C 180,E1 -9228.05,E2 -9228.05} C_VEL
LIN {X 0,Y 444.085,Z 682.895,A -85,B 0,C 180,E1 -9229.098,E2 -9229.098} C_VEL
LIN {X 0,Y 442.987,Z 695.291,A -85,B 0,C 180,E1 -9230.316,E2 -9230.316} C_VEL
LIN {X 0,Y 441.997,Z 706.767,A -85,B 0,C 180,E1 -9231.676,E2 -9231.676} C_VEL
LIN {X 0,Y 441.059,Z 716.51,A -85,B 0,C 180,E1 -9233.043,E2 -9233.043} C_VEL
LIN {X 0,Y 440.243,Z 726.342,A -85,B 0,C 180,E1 -9234.699,E2 -9234.699} C_VEL
LIN {X 0,Y 439.654,Z 733.941,A -85,B 0,C 180,E1 -9236.226,E2 -9236.226} C_VEL
LIN {X 0,Y 439.04,Z 741.626,A -85,B 0,C 180,E1 -9238.114,E2 -9238.114} C_VEL
LIN {X 0,Y 438.736,Z 747.376,A -85,B 0,C 180,E1 -9239.885,E2 -9239.885} C_VEL
LIN {X 0,Y 438.411,Z 752.176,A -85,B 0,C 180,E1 -9241.802,E2 -9241.802} C_VEL
LIN {X 0,Y 437.646,Z 753.746,A -85,B 0,C 180,E1 -9242.539,E2 -9242.539} C_VEL
LIN {X 0,Y 434.647,Z 755.83,A -85,B 0,C 180,E1 -9243.749,E2 -9243.749} C_VEL
LIN {X 0,Y 432.162,Z 757.143,A -85,B 0,C 180,E1 -9244.737,E2 -9244.737} C_VEL
LIN {X 0,Y 431.112,Z 757.888,A -85,B 0,C 180,E1 -9245.506,E2 -9245.506} C_VEL
LIN {X 0,Y 431.033,Z 758.106,A -85,B 0,C 180,E1 -9245.767,E2 -9245.767} C_VEL
LIN {X 0,Y 430.999,Z 758.77,A -85,B 0,C 180,E1 -9246.962,E2 -9246.962} C_VEL
LIN {X 0,Y 431.042,Z 758.792,A -85,B 0,C 180,E1 -9248.98,E2 -9248.98} C_VEL
LIN {X 0,Y 431.1,Z 757.491,A -85,B 0,C 180,E1 -9251.005,E2 -9251.005} C_VEL
LIN {X 0,Y 431.206,Z 754.978,A -85,B 0,C 180,E1 -9252.941,E2 -9252.941} C_VEL
LIN {X 0,Y 431.49,Z 751.134,A -85,B 0,C 180,E1 -9254.895,E2 -9254.895} C_VEL
LIN {X 0,Y 431.729,Z 745.972,A -85,B 0,C 180,E1 -9256.827,E2 -9256.827} C_VEL
LIN {X 0,Y 432.209,Z 739.348,A -85,B 0,C 180,E1 -9258.748,E2 -9258.748} C_VEL
LIN {X 0,Y 432.742,Z 732.231,A -85,B 0,C 180,E1 -9260.418,E2 -9260.418} C_VEL
LIN {X 0,Y 433.565,Z 723.296,A -85,B 0,C 180,E1 -9262.146,E2 -9262.146} C_VEL
LIN {X 0,Y 434.434,Z 713.427,A -85,B 0,C 180,E1 -9263.732,E2 -9263.732} C_VEL
LIN {X 0,Y 435.447,Z 702.948,A -85,B 0,C 180,E1 -9265.14,E2 -9265.14} C_VEL
LIN {X 0,Y 436.46,Z 691.552,A -85,B 0,C 180,E1 -9266.429,E2 -9266.429} C_VEL
LIN {X 0,Y 437.543,Z 679.301,A -85,B 0,C 180,E1 -9267.584,E2 -9267.584} C_VEL
LIN {X 0,Y 438.662,Z 665.832,A -85,B 0,C 180,E1 -9268.623,E2 -9268.623} C_VEL
LIN {X 0,Y 439.581,Z 651.98,A -85,B 0,C 180,E1 -9269.485,E2 -9269.485} C_VEL
LIN {X 0,Y 440.486,Z 636.333,A -85,B 0,C 180,E1 -9270.229,E2 -9270.229} C_VEL
LIN {X 0,Y 441.103,Z 621.467,A -85,B 0,C 180,E1 -9270.742,E2 -9270.742} C_VEL
LIN {X 0,Y 441.497,Z 606.182,A -85,B 0,C 180,E1 -9271.084,E2 -9271.084} C_VEL
LIN {X 0,Y 443.61,Z 474.399,A -85,B 0,C 180,E1 -9273.282,E2 -9273.282} C_VEL
LIN {X 0,Y 440.731,Z 462.487,A -85,B 0,C 180,E1 -9273.67,E2 -9273.67} C_VEL
LIN {X 0,Y 436.021,Z 451.229,A -85,B 0,C 180,E1 -9274.168,E2 -9274.168} C_VEL
LIN {X 0,Y 435.195,Z 449.146,A -85,B 0,C 180,E1 -9274.267,E2 -9274.267} C_VEL
LIN {X 0,Y 432.53,Z 437.234,A -85,B 0,C 180,E1 -9276.766,E2 -9276.766} C_VEL
LIN {X 0,Y 432.449,Z 437.247,A -85,B 0,C 180,E1 -9279.353,E2 -9279.353} C_VEL
LIN {X 0,Y 432.449,Z 437.243,A -85,B 0,C 180,E1 -9282.812,E2 -9282.812} C_VEL
LIN {X 0,Y 432.417,Z 437.245,A -85,B 0,C 180,E1 -9286.479,E2 -9286.479} C_VEL
LIN {X 0,Y 432.377,Z 437.251,A -85,B 0,C 180,E1 -9289.959,E2 -9289.959} C_VEL
LIN {X 0,Y 432.324,Z 437.257,A -85,B 0,C 180,E1 -9292.964,E2 -9292.964} C_VEL
LIN {X 0,Y 432.369,Z 437.252,A -85,B 0,C 180,E1 -9296.032,E2 -9296.032} C_VEL
LIN {X 0,Y 432.352,Z 437.25,A -85,B 0,C 180,E1 -9299.187,E2 -9299.187} C_VEL
LIN {X 0,Y 432.329,Z 437.247,A -85,B 0,C 180,E1 -9302.293,E2 -9302.293} C_VEL
LIN {X 0,Y 432.344,Z 437.253,A -85,B 0,C 180,E1 -9304.677,E2 -9304.677} C_VEL
LIN {X 0,Y 432.35,Z 437.246,A -85,B 0,C 180,E1 -9308.149,E2 -9308.149} C_VEL
LIN {X 0,Y 432.365,Z 437.254,A -85,B 0,C 180,E1 -9311.606,E2 -9311.606} C_VEL
LIN {X 0,Y 432.343,Z 437.251,A -85,B 0,C 180,E1 -9314.346,E2 -9314.346} C_VEL
LIN {X 0,Y 432.322,Z 437.255,A -85,B 0,C 180,E1 -9317.015,E2 -9317.015} C_VEL
LIN {X 0,Y 432.358,Z 437.254,A -85,B 0,C 180,E1 -9319.817,E2 -9319.817} C_VEL
LIN {X 0,Y 432.318,Z 437.254,A -85,B 0,C 180,E1 -9323.023,E2 -9323.023} C_VEL
LIN {X 0,Y 432.361,Z 437.253,A -85,B 0,C 180,E1 -9325.996,E2 -9325.996} C_VEL
LIN {X 0,Y 432.348,Z 437.25,A -85,B 0,C 180,E1 -9329.489,E2 -9329.489} C_VEL
LIN {X 0,Y 432.394,Z 437.246,A -85,B 0,C 180,E1 -9332.928,E2 -9332.928} C_VEL
LIN {X 0,Y 432.372,Z 437.24,A -85,B 0,C 180,E1 -9336.023,E2 -9336.023} C_VEL
LIN {X 0,Y 432.351,Z 437.25,A -85,B 0,C 180,E1 -9339.046,E2 -9339.046} C_VEL
LIN {X 0,Y 432.379,Z 437.244,A -85,B 0,C 180,E1 -9342.011,E2 -9342.011} C_VEL
LIN {X 0,Y 432.396,Z 437.24,A -85,B 0,C 180,E1 -9344.926,E2 -9344.926} C_VEL
LIN {X 0,Y 432.459,Z 437.24,A -85,B 0,C 180,E1 -9347.803,E2 -9347.803} C_VEL
LIN {X 0,Y 432.492,Z 437.23,A -85,B 0,C 180,E1 -9351.59,E2 -9351.59} C_VEL
LIN {X 0,Y 432.598,Z 437.22,A -85,B 0,C 180,E1 -9354.406,E2 -9354.406} C_VEL
LIN {X 0,Y 432.604,Z 437.218,A -85,B 0,C 180,E1 -9358.138,E2 -9358.138} C_VEL
LIN {X 0,Y 432.733,Z 437.207,A -85,B 0,C 180,E1 -9360,E2 -9360} C_VEL
LIN {X 0,Y 432.605,Z 437.215,A -85,B 0,C 180,E1 -9362.793,E2 -9362.793} C_VEL
LIN {X 0,Y 432.572,Z 437.22,A -85,B 0,C 180,E1 -9366.53,E2 -9366.53} C_VEL
LIN {X 0,Y 432.442,Z 437.243,A -85,B 0,C 180,E1 -9369.353,E2 -9369.353} C_VEL
LIN {X 0,Y 432.43,Z 437.232,A -85,B 0,C 180,E1 -9372.803,E2 -9372.803} C_VEL
LIN {X 0,Y 432.412,Z 437.242,A -85,B 0,C 180,E1 -9376.479,E2 -9376.479} C_VEL
LIN {X 0,Y 432.339,Z 437.255,A -85,B 0,C 180,E1 -9379.96,E2 -9379.96} C_VEL
LIN {X 0,Y 432.319,Z 437.254,A -85,B 0,C 180,E1 -9382.964,E2 -9382.964} C_VEL
LIN {X 0,Y 432.364,Z 437.253,A -85,B 0,C 180,E1 -9386.032,E2 -9386.032} C_VEL
LIN {X 0,Y 432.348,Z 437.252,A -85,B 0,C 180,E1 -9389.187,E2 -9389.187} C_VEL
LIN {X 0,Y 432.324,Z 437.256,A -85,B 0,C 180,E1 -9392.293,E2 -9392.293} C_VEL
LIN {X 0,Y 432.341,Z 437.253,A -85,B 0,C 180,E1 -9394.677,E2 -9394.677} C_VEL
LIN {X 0,Y 432.347,Z 437.254,A -85,B 0,C 180,E1 -9398.149,E2 -9398.149} C_VEL
LIN {X 0,Y 432.333,Z 437.26,A -85,B 0,C 180,E1 -9401.602,E2 -9401.602} C_VEL
LIN {X 0,Y 432.333,Z 437.255,A -85,B 0,C 180,E1 -9404.347,E2 -9404.347} C_VEL
LIN {X 0,Y 432.366,Z 437.251,A -85,B 0,C 180,E1 -9407.009,E2 -9407.009} C_VEL
LIN {X 0,Y 432.335,Z 437.258,A -85,B 0,C 180,E1 -9409.82,E2 -9409.82} C_VEL
LIN {X 0,Y 432.306,Z 437.257,A -85,B 0,C 180,E1 -9413.022,E2 -9413.022} C_VEL
LIN {X 0,Y 432.359,Z 437.253,A -85,B 0,C 180,E1 -9415.996,E2 -9415.996} C_VEL
LIN {X 0,Y 432.322,Z 437.303,A -85,B 0,C 180,E1 -9417.762,E2 -9417.762} C_VEL
LIN {X 0,Y 436,Z 451.768,A -85,B 0,C 180,E1 -9420.51,E2 -9420.51} C_VEL
LIN {X 0,Y 438.145,Z 461.532,A -85,B 0,C 180,E1 -9422.279,E2 -9422.279} C_VEL
LIN {X 0,Y 437.504,Z 471.904,A -85,B 0,C 180,E1 -9423.919,E2 -9423.919} C_VEL
LIN {X 0,Y 443.244,Z 501.231,A -85,B 0,C 180,E1 -9424.792,E2 -9424.792} C_VEL
LIN {X 0,Y 441.774,Z 601.448,A -85,B 0,C 180,E1 -9426.471,E2 -9426.471} C_VEL
LIN {X 0,Y 441.157,Z 638.764,A -85,B 0,C 180,E1 -9427.119,E2 -9427.119} C_VEL
LIN {X 0,Y 440.457,Z 654.457,A -85,B 0,C 180,E1 -9427.57,E2 -9427.57} C_VEL
LIN {X 0,Y 439.628,Z 669.839,A -85,B 0,C 180,E1 -9428.216,E2 -9428.216} C_VEL
LIN {X 0,Y 438.648,Z 683.896,A -85,B 0,C 180,E1 -9428.992,E2 -9428.992} C_VEL
LIN {X 0,Y 437.629,Z 697.266,A -85,B 0,C 180,E1 -9429.924,E2 -9429.924} C_VEL
LIN {X 0,Y 436.398,Z 710.863,A -85,B 0,C 180,E1 -9431.088,E2 -9431.088} C_VEL
LIN {X 0,Y 435.258,Z 723.787,A -85,B 0,C 180,E1 -9432.446,E2 -9432.446} C_VEL
LIN {X 0,Y 434.3,Z 734.49,A -85,B 0,C 180,E1 -9433.79,E2 -9433.79} C_VEL
LIN {X 0,Y 433.323,Z 745.436,A -85,B 0,C 180,E1 -9435.44,E2 -9435.44} C_VEL
LIN {X 0,Y 432.432,Z 755.054,A -85,B 0,C 180,E1 -9437.196,E2 -9437.196} C_VEL
LIN {X 0,Y 432.117,Z 762.083,A -85,B 0,C 180,E1 -9438.745,E2 -9438.745} C_VEL
LIN {X 0,Y 431.606,Z 769.127,A -85,B 0,C 180,E1 -9440.628,E2 -9440.628} C_VEL
LIN {X 0,Y 431.387,Z 774.669,A -85,B 0,C 180,E1 -9442.511,E2 -9442.511} C_VEL
LIN {X 0,Y 431.231,Z 778.857,A -85,B 0,C 180,E1 -9444.388,E2 -9444.388} C_VEL
LIN {X 0,Y 431.148,Z 781.792,A -85,B 0,C 180,E1 -9446.261,E2 -9446.261} C_VEL
LIN {X 0,Y 431.195,Z 783.544,A -85,B 0,C 180,E1 -9448.131,E2 -9448.131} C_VEL
LIN {X 0,Y 431.164,Z 784.138,A -85,B 0,C 180,E1 -9449.999,E2 -9449.999} C_VEL
LIN {X 0,Y 431.195,Z 783.532,A -85,B 0,C 180,E1 -9451.868,E2 -9451.868} C_VEL
LIN {X 0,Y 431.166,Z 781.773,A -85,B 0,C 180,E1 -9453.738,E2 -9453.738} C_VEL
LIN {X 0,Y 431.236,Z 778.837,A -85,B 0,C 180,E1 -9455.611,E2 -9455.611} C_VEL
LIN {X 0,Y 431.387,Z 774.655,A -85,B 0,C 180,E1 -9457.488,E2 -9457.488} C_VEL
LIN {X 0,Y 431.605,Z 769.113,A -85,B 0,C 180,E1 -9459.371,E2 -9459.371} C_VEL
LIN {X 0,Y 432.113,Z 762.07,A -85,B 0,C 180,E1 -9461.254,E2 -9461.254} C_VEL
LIN {X 0,Y 432.667,Z 753.304,A -85,B 0,C 180,E1 -9463.144,E2 -9463.144} C_VEL
LIN {X 0,Y 433.428,Z 743.998,A -85,B 0,C 180,E1 -9464.796,E2 -9464.796} C_VEL
LIN {X 0,Y 434.252,Z 734.542,A -85,B 0,C 180,E1 -9466.21,E2 -9466.21} C_VEL
LIN {X 0,Y 435.325,Z 723.553,A -85,B 0,C 180,E1 -9467.591,E2 -9467.591} C_VEL
LIN {X 0,Y 436.397,Z 711.037,A -85,B 0,C 180,E1 -9468.911,E2 -9468.911} C_VEL
LIN {X 0,Y 437.614,Z 697.536,A -85,B 0,C 180,E1 -9470.076,E2 -9470.076} C_VEL
LIN {X 0,Y 438.675,Z 684.281,A -85,B 0,C 180,E1 -9471.005,E2 -9471.005} C_VEL
LIN {X 0,Y 439.661,Z 670.491,A -85,B 0,C 180,E1 -9471.779,E2 -9471.779} C_VEL
LIN {X 0,Y 440.475,Z 655.693,A -85,B 0,C 180,E1 -9472.417,E2 -9472.417} C_VEL
LIN {X 0,Y 441.167,Z 640.373,A -85,B 0,C 180,E1 -9472.879,E2 -9472.879} C_VEL
LIN {X 0,Y 441.68,Z 616.613,A -85,B 0,C 180,E1 -9473.316,E2 -9473.316} C_VEL
LIN {X 0,Y 443.53,Z 502.216,A -85,B 0,C 180,E1 -9475.23,E2 -9475.23} C_VEL
LIN {X 0,Y 438.313,Z 475.103,A -85,B 0,C 180,E1 -9476.05,E2 -9476.05} C_VEL
LIN {X 0,Y 437.511,Z 471.222,A -85,B 0,C 180,E1 -9476.182,E2 -9476.182} C_VEL
LIN {X 0,Y 438.218,Z 461.673,A -85,B 0,C 180,E1 -9477.715,E2 -9477.715} C_VEL
LIN {X 0,Y 435.403,Z 449.154,A -85,B 0,C 180,E1 -9480.024,E2 -9480.024} C_VEL
LIN {X 0,Y 432.33,Z 437.26,A -85,B 0,C 180,E1 -9482.383,E2 -9482.383} C_VEL
LIN {X 0,Y 432.341,Z 437.253,A -85,B 0,C 180,E1 -9485.631,E2 -9485.631} C_VEL
LIN {X 0,Y 432.357,Z 437.255,A -85,B 0,C 180,E1 -9488.717,E2 -9488.717} C_VEL
LIN {X 0,Y 432.369,Z 437.254,A -85,B 0,C 180,E1 -9491.792,E2 -9491.792} C_VEL
LIN {X 0,Y 432.373,Z 437.255,A -85,B 0,C 180,E1 -9494.341,E2 -9494.341} C_VEL
LIN {X 0,Y 432.328,Z 437.259,A -85,B 0,C 180,E1 -9498.202,E2 -9498.202} C_VEL
LIN {X 0,Y 432.346,Z 437.253,A -85,B 0,C 180,E1 -9501.283,E2 -9501.283} C_VEL
LIN {X 0,Y 432.339,Z 437.256,A -85,B 0,C 180,E1 -9504.367,E2 -9504.367} C_VEL
LIN {X 0,Y 432.316,Z 437.254,A -85,B 0,C 180,E1 -9507.557,E2 -9507.557} C_VEL
LIN {X 0,Y 432.336,Z 437.256,A -85,B 0,C 180,E1 -9510.812,E2 -9510.812} C_VEL
LIN {X 0,Y 432.358,Z 437.251,A -85,B 0,C 180,E1 -9513.967,E2 -9513.967} C_VEL
LIN {X 0,Y 432.312,Z 437.257,A -85,B 0,C 180,E1 -9517.036,E2 -9517.036} C_VEL
LIN {X 0,Y 432.379,Z 437.252,A -85,B 0,C 180,E1 -9520.514,E2 -9520.514} C_VEL
LIN {X 0,Y 432.423,Z 437.241,A -85,B 0,C 180,E1 -9523.961,E2 -9523.961} C_VEL
LIN {X 0,Y 432.473,Z 437.235,A -85,B 0,C 180,E1 -9527.804,E2 -9527.804} C_VEL
LIN {X 0,Y 432.484,Z 437.234,A -85,B 0,C 180,E1 -9531.59,E2 -9531.59} C_VEL
LIN {X 0,Y 432.591,Z 437.222,A -85,B 0,C 180,E1 -9534.406,E2 -9534.406} C_VEL
LIN {X 0,Y 432.599,Z 437.22,A -85,B 0,C 180,E1 -9538.138,E2 -9538.138} C_VEL
LIN {X 0,Y 432.726,Z 437.208,A -85,B 0,C 180,E1 -9540,E2 -9540} C_VEL
LIN {X 0,Y 432.599,Z 437.224,A -85,B 0,C 180,E1 -9542.794,E2 -9542.794} C_VEL
LIN {X 0,Y 432.566,Z 437.229,A -85,B 0,C 180,E1 -9546.531,E2 -9546.531} C_VEL
LIN {X 0,Y 432.436,Z 437.241,A -85,B 0,C 180,E1 -9549.354,E2 -9549.354} C_VEL
LIN {X 0,Y 432.424,Z 437.245,A -85,B 0,C 180,E1 -9552.804,E2 -9552.804} C_VEL
LIN {X 0,Y 432.416,Z 437.246,A -85,B 0,C 180,E1 -9556.484,E2 -9556.484} C_VEL
LIN {X 0,Y 432.333,Z 437.256,A -85,B 0,C 180,E1 -9559.961,E2 -9559.961} C_VEL
LIN {X 0,Y 432.313,Z 437.26,A -85,B 0,C 180,E1 -9562.965,E2 -9562.965} C_VEL
LIN {X 0,Y 432.359,Z 437.252,A -85,B 0,C 180,E1 -9566.033,E2 -9566.033} C_VEL
LIN {X 0,Y 432.347,Z 437.253,A -85,B 0,C 180,E1 -9569.187,E2 -9569.187} C_VEL
LIN {X 0,Y 432.327,Z 437.256,A -85,B 0,C 180,E1 -9572.295,E2 -9572.295} C_VEL
LIN {X 0,Y 432.337,Z 437.255,A -85,B 0,C 180,E1 -9574.678,E2 -9574.678} C_VEL
LIN {X 0,Y 432.349,Z 437.259,A -85,B 0,C 180,E1 -9578.149,E2 -9578.149} C_VEL
LIN {X 0,Y 432.39,Z 437.271,A -85,B 0,C 180,E1 -9579.097,E2 -9579.097} C_VEL
LIN {X 0,Y 435.367,Z 449.66,A -85,B 0,C 180,E1 -9581.738,E2 -9581.738} C_VEL
LIN {X 0,Y 441.51,Z 464.395,A -85,B 0,C 180,E1 -9582.418,E2 -9582.418} C_VEL
LIN {X 0,Y 443.891,Z 475.592,A -85,B 0,C 180,E1 -9582.772,E2 -9582.772} C_VEL
LIN {X 0,Y 441.533,Z 614.686,A -85,B 0,C 180,E1 -9585.125,E2 -9585.125} C_VEL
LIN {X 0,Y 440.906,Z 630.453,A -85,B 0,C 180,E1 -9585.58,E2 -9585.58} C_VEL
LIN {X 0,Y 440.161,Z 645.177,A -85,B 0,C 180,E1 -9586.197,E2 -9586.197} C_VEL
LIN {X 0,Y 439.292,Z 658.958,A -85,B 0,C 180,E1 -9586.959,E2 -9586.959} C_VEL
LIN {X 0,Y 438.187,Z 673.365,A -85,B 0,C 180,E1 -9587.963,E2 -9587.963} C_VEL
LIN {X 0,Y 437.109,Z 686.334,A -85,B 0,C 180,E1 -9589.086,E2 -9589.086} C_VEL
LIN {X 0,Y 435.963,Z 698.568,A -85,B 0,C 180,E1 -9590.367,E2 -9590.367} C_VEL
LIN {X 0,Y 434.873,Z 710.074,A -85,B 0,C 180,E1 -9591.819,E2 -9591.819} C_VEL
LIN {X 0,Y 433.835,Z 720.817,A -85,B 0,C 180,E1 -9593.455,E2 -9593.455} C_VEL
LIN {X 0,Y 432.977,Z 729.779,A -85,B 0,C 180,E1 -9595.099,E2 -9595.099} C_VEL
LIN {X 0,Y 432.3,Z 738.262,A -85,B 0,C 180,E1 -9597.003,E2 -9597.003} C_VEL
LIN {X 0,Y 431.865,Z 744.114,A -85,B 0,C 180,E1 -9598.618,E2 -9598.618} C_VEL
LIN {X 0,Y 431.608,Z 748.857,A -85,B 0,C 180,E1 -9600.223,E2 -9600.223} C_VEL
LIN {X 0,Y 431.326,Z 752.621,A -85,B 0,C 180,E1 -9601.803,E2 -9601.803} C_VEL
LIN {X 0,Y 431.13,Z 756.177,A -85,B 0,C 180,E1 -9603.888,E2 -9603.888} C_VEL
LIN {X 0,Y 431.033,Z 758.106,A -85,B 0,C 180,E1 -9605.767,E2 -9605.767} C_VEL
LIN {X 0,Y 430.375,Z 758.661,A -85,B 0,C 180,E1 -9606.544,E2 -9606.544} C_VEL
LIN {X 0,Y 427.497,Z 759.114,A -85,B 0,C 180,E1 -9607.811,E2 -9607.811} C_VEL
LIN {X 0,Y 425.059,Z 759.033,A -85,B 0,C 180,E1 -9608.834,E2 -9608.834} C_VEL
LIN {X 0,Y 424.02,Z 758.713,A -85,B 0,C 180,E1 -9609.625,E2 -9609.625} C_VEL
LIN {X 0,Y 423.94,Z 758.539,A -85,B 0,C 180,E1 -9609.892,E2 -9609.892} C_VEL
LIN {X 0,Y 424.04,Z 757.054,A -85,B 0,C 180,E1 -9611.646,E2 -9611.646} C_VEL
LIN {X 0,Y 424.22,Z 754.119,A -85,B 0,C 180,E1 -9613.643,E2 -9613.643} C_VEL
LIN {X 0,Y 424.482,Z 749.881,A -85,B 0,C 180,E1 -9615.621,E2 -9615.621} C_VEL
LIN {X 0,Y 424.85,Z 744.275,A -85,B 0,C 180,E1 -9617.582,E2 -9617.582} C_VEL
LIN {X 0,Y 425.413,Z 737.16,A -85,B 0,C 180,E1 -9619.53,E2 -9619.53} C_VEL
LIN {X 0,Y 426.026,Z 729.584,A -85,B 0,C 180,E1 -9621.223,E2 -9621.223} C_VEL
LIN {X 0,Y 426.887,Z 720.466,A -85,B 0,C 180,E1 -9622.908,E2 -9622.908} C_VEL
LIN {X 0,Y 427.981,Z 709.476,A -85,B 0,C 180,E1 -9624.583,E2 -9624.583} C_VEL
LIN {X 0,Y 429.084,Z 698.217,A -85,B 0,C 180,E1 -9626.009,E2 -9626.009} C_VEL
LIN {X 0,Y 430.243,Z 685.88,A -85,B 0,C 180,E1 -9627.309,E2 -9627.309} C_VEL
LIN {X 0,Y 431.471,Z 672.253,A -85,B 0,C 180,E1 -9628.484,E2 -9628.484} C_VEL
LIN {X 0,Y 432.524,Z 658.914,A -85,B 0,C 180,E1 -9629.419,E2 -9629.419} C_VEL
LIN {X 0,Y 433.476,Z 644.179,A -85,B 0,C 180,E1 -9630.233,E2 -9630.233} C_VEL
LIN {X 0,Y 434.261,Z 628.709,A -85,B 0,C 180,E1 -9630.87,E2 -9630.87} C_VEL
LIN {X 0,Y 434.833,Z 613.303,A -85,B 0,C 180,E1 -9631.303,E2 -9631.303} C_VEL
LIN {X 0,Y 437.127,Z 475.355,A -85,B 0,C 180,E1 -9633.661,E2 -9633.661} C_VEL
LIN {X 0,Y 434.644,Z 465.114,A -85,B 0,C 180,E1 -9634.003,E2 -9634.003} C_VEL
LIN {X 0,Y 429.035,Z 451.911,A -85,B 0,C 180,E1 -9634.607,E2 -9634.607} C_VEL
LIN {X 0,Y 428.002,Z 449.287,A -85,B 0,C 180,E1 -9634.739,E2 -9634.739} C_VEL
LIN {X 0,Y 425.461,Z 438.114,A -85,B 0,C 180,E1 -9637.112,E2 -9637.112} C_VEL
LIN {X 0,Y 425.377,Z 438.113,A -85,B 0,C 180,E1 -9640.472,E2 -9640.472} C_VEL
LIN {X 0,Y 425.388,Z 438.123,A -85,B 0,C 180,E1 -9643.374,E2 -9643.374} C_VEL
LIN {X 0,Y 425.366,Z 438.123,A -85,B 0,C 180,E1 -9646.605,E2 -9646.605} C_VEL
LIN {X 0,Y 425.365,Z 438.129,A -85,B 0,C 180,E1 -9649.648,E2 -9649.648} C_VEL
LIN {X 0,Y 425.312,Z 438.134,A -85,B 0,C 180,E1 -9653.365,E2 -9653.365} C_VEL
LIN {X 0,Y 425.352,Z 438.124,A -85,B 0,C 180,E1 -9656.844,E2 -9656.844} C_VEL
LIN {X 0,Y 425.319,Z 438.132,A -85,B 0,C 180,E1 -9659.718,E2 -9659.718} C_VEL
LIN {X 0,Y 425.285,Z 438.124,A -85,B 0,C 180,E1 -9663.048,E2 -9663.048} C_VEL
LIN {X 0,Y 425.288,Z 438.133,A -85,B 0,C 180,E1 -9665.929,E2 -9665.929} C_VEL
LIN {X 0,Y 425.306,Z 438.123,A -85,B 0,C 180,E1 -9669.044,E2 -9669.044} C_VEL
LIN {X 0,Y 425.295,Z 438.13,A -85,B 0,C 180,E1 -9671.958,E2 -9671.958} C_VEL
LIN {X 0,Y 425.289,Z 438.133,A -85,B 0,C 180,E1 -9675.283,E2 -9675.283} C_VEL
LIN {X 0,Y 425.306,Z 438.121,A -85,B 0,C 180,E1 -9678.625,E2 -9678.625} C_VEL
LIN {X 0,Y 425.324,Z 438.128,A -85,B 0,C 180,E1 -9681.104,E2 -9681.104} C_VEL
LIN {X 0,Y 425.302,Z 438.123,A -85,B 0,C 180,E1 -9684.664,E2 -9684.664} C_VEL
LIN {X 0,Y 425.266,Z 438.133,A -85,B 0,C 180,E1 -9688.073,E2 -9688.073} C_VEL
LIN {X 0,Y 425.332,Z 438.121,A -85,B 0,C 180,E1 -9691.368,E2 -9691.368} C_VEL
LIN {X 0,Y 425.296,Z 438.128,A -85,B 0,C 180,E1 -9694.554,E2 -9694.554} C_VEL
LIN {X 0,Y 425.289,Z 438.126,A -85,B 0,C 180,E1 -9697.661,E2 -9697.661} C_VEL
LIN {X 0,Y 425.363,Z 438.121,A -85,B 0,C 180,E1 -9700.704,E2 -9700.704} C_VEL
LIN {X 0,Y 425.389,Z 438.112,A -85,B 0,C 180,E1 -9703.688,E2 -9703.688} C_VEL
LIN {X 0,Y 425.412,Z 438.121,A -85,B 0,C 180,E1 -9707.598,E2 -9707.598} C_VEL
LIN {X 0,Y 425.443,Z 438.106,A -85,B 0,C 180,E1 -9711.45,E2 -9711.45} C_VEL
LIN {X 0,Y 425.554,Z 438.097,A -85,B 0,C 180,E1 -9714.313,E2 -9714.313} C_VEL
LIN {X 0,Y 425.573,Z 438.094,A -85,B 0,C 180,E1 -9718.107,E2 -9718.107} C_VEL
LIN {X 0,Y 425.703,Z 438.083,A -85,B 0,C 180,E1 -9720,E2 -9720} C_VEL
LIN {X 0,Y 425.556,Z 438.093,A -85,B 0,C 180,E1 -9722.84,E2 -9722.84} C_VEL
LIN {X 0,Y 425.53,Z 438.097,A -85,B 0,C 180,E1 -9726.639,E2 -9726.639} C_VEL
LIN {X 0,Y 425.401,Z 438.122,A -85,B 0,C 180,E1 -9729.509,E2 -9729.509} C_VEL
LIN {X 0,Y 425.393,Z 438.109,A -85,B 0,C 180,E1 -9732.903,E2 -9732.903} C_VEL
LIN {X 0,Y 425.361,Z 438.12,A -85,B 0,C 180,E1 -9736.605,E2 -9736.605} C_VEL
LIN {X 0,Y 425.328,Z 438.122,A -85,B 0,C 180,E1 -9739.635,E2 -9739.635} C_VEL
LIN {X 0,Y 425.307,Z 438.131,A -85,B 0,C 180,E1 -9743.365,E2 -9743.365} C_VEL
LIN {X 0,Y 425.348,Z 438.124,A -85,B 0,C 180,E1 -9746.844,E2 -9746.844} C_VEL
LIN {X 0,Y 425.315,Z 438.134,A -85,B 0,C 180,E1 -9749.717,E2 -9749.717} C_VEL
LIN {X 0,Y 425.282,Z 438.132,A -85,B 0,C 180,E1 -9753.048,E2 -9753.048} C_VEL
LIN {X 0,Y 425.284,Z 438.135,A -85,B 0,C 180,E1 -9755.929,E2 -9755.929} C_VEL
LIN {X 0,Y 425.303,Z 438.13,A -85,B 0,C 180,E1 -9759.044,E2 -9759.044} C_VEL
LIN {X 0,Y 425.276,Z 438.133,A -85,B 0,C 180,E1 -9762.653,E2 -9762.653} C_VEL
LIN {X 0,Y 425.319,Z 438.131,A -85,B 0,C 180,E1 -9766.051,E2 -9766.051} C_VEL
LIN {X 0,Y 425.302,Z 438.131,A -85,B 0,C 180,E1 -9768.625,E2 -9768.625} C_VEL
LIN {X 0,Y 425.306,Z 438.132,A -85,B 0,C 180,E1 -9771.102,E2 -9771.102} C_VEL
LIN {X 0,Y 425.299,Z 438.136,A -85,B 0,C 180,E1 -9774.664,E2 -9774.664} C_VEL
LIN {X 0,Y 425.291,Z 438.234,A -85,B 0,C 180,E1 -9777.381,E2 -9777.381} C_VEL
LIN {X 0,Y 429.051,Z 453.012,A -85,B 0,C 180,E1 -9780.245,E2 -9780.245} C_VEL
LIN {X 0,Y 431.341,Z 463.298,A -85,B 0,C 180,E1 -9782.144,E2 -9782.144} C_VEL
LIN {X 0,Y 430.789,Z 471.526,A -85,B 0,C 180,E1 -9783.483,E2 -9783.483} C_VEL
LIN {X 0,Y 436.857,Z 502.838,A -85,B 0,C 180,E1 -9784.438,E2 -9784.438} C_VEL
LIN {X 0,Y 435.114,Z 607.793,A -85,B 0,C 180,E1 -9786.215,E2 -9786.215} C_VEL
LIN {X 0,Y 434.568,Z 639.324,A -85,B 0,C 180,E1 -9786.784,E2 -9786.784} C_VEL
LIN {X 0,Y 433.832,Z 654.767,A -85,B 0,C 180,E1 -9787.24,E2 -9787.24} C_VEL
LIN {X 0,Y 432.984,Z 670.039,A -85,B 0,C 180,E1 -9787.897,E2 -9787.897} C_VEL
LIN {X 0,Y 432,Z 683.544,A -85,B 0,C 180,E1 -9788.653,E2 -9788.653} C_VEL
LIN {X 0,Y 430.922,Z 696.944,A -85,B 0,C 180,E1 -9789.597,E2 -9789.597} C_VEL
LIN {X 0,Y 429.617,Z 710.572,A -85,B 0,C 180,E1 -9790.778,E2 -9790.778} C_VEL
LIN {X 0,Y 428.428,Z 722.82,A -85,B 0,C 180,E1 -9792.071,E2 -9792.071} C_VEL
LIN {X 0,Y 427.398,Z 734.236,A -85,B 0,C 180,E1 -9793.521,E2 -9793.521} C_VEL
LIN {X 0,Y 426.371,Z 745.194,A -85,B 0,C 180,E1 -9795.197,E2 -9795.197} C_VEL
LIN {X 0,Y 425.474,Z 754.704,A -85,B 0,C 180,E1 -9796.957,E2 -9796.957} C_VEL
LIN {X 0,Y 425.103,Z 761.853,A -85,B 0,C 180,E1 -9798.557,E2 -9798.557} C_VEL
LIN {X 0,Y 424.538,Z 768.902,A -85,B 0,C 180,E1 -9800.471,E2 -9800.471} C_VEL
LIN {X 0,Y 424.31,Z 774.449,A -85,B 0,C 180,E1 -9802.385,E2 -9802.385} C_VEL
LIN {X 0,Y 424.146,Z 778.641,A -85,B 0,C 180,E1 -9804.294,E2 -9804.294} C_VEL
LIN {X 0,Y 424.06,Z 781.58,A -85,B 0,C 180,E1 -9806.198,E2 -9806.198} C_VEL
LIN {X 0,Y 424.12,Z 783.336,A -85,B 0,C 180,E1 -9808.1,E2 -9808.1} C_VEL
LIN {X 0,Y 424.081,Z 783.931,A -85,B 0,C 180,E1 -9809.999,E2 -9809.999} C_VEL
LIN {X 0,Y 424.121,Z 783.326,A -85,B 0,C 180,E1 -9811.899,E2 -9811.899} C_VEL
LIN {X 0,Y 424.076,Z 781.568,A -85,B 0,C 180,E1 -9813.8,E2 -9813.8} C_VEL
LIN {X 0,Y 424.151,Z 778.633,A -85,B 0,C 180,E1 -9815.705,E2 -9815.705} C_VEL
LIN {X 0,Y 424.309,Z 774.45,A -85,B 0,C 180,E1 -9817.614,E2 -9817.614} C_VEL
LIN {X 0,Y 424.537,Z 768.909,A -85,B 0,C 180,E1 -9819.528,E2 -9819.528} C_VEL
LIN {X 0,Y 425.101,Z 761.865,A -85,B 0,C 180,E1 -9821.442,E2 -9821.442} C_VEL
LIN {X 0,Y 425.68,Z 753.103,A -85,B 0,C 180,E1 -9823.364,E2 -9823.364} C_VEL
LIN {X 0,Y 426.484,Z 743.805,A -85,B 0,C 180,E1 -9825.042,E2 -9825.042} C_VEL
LIN {X 0,Y 427.381,Z 734.358,A -85,B 0,C 180,E1 -9826.478,E2 -9826.478} C_VEL
LIN {X 0,Y 428.563,Z 722.508,A -85,B 0,C 180,E1 -9827.985,E2 -9827.985} C_VEL
LIN {X 0,Y 429.77,Z 709.636,A -85,B 0,C 180,E1 -9829.338,E2 -9829.338} C_VEL
LIN {X 0,Y 431.047,Z 695.84,A -85,B 0,C 180,E1 -9830.52,E2 -9830.52} C_VEL
LIN {X 0,Y 432.179,Z 682.301,A -85,B 0,C 180,E1 -9831.462,E2 -9831.462} C_VEL
LIN {X 0,Y 433.22,Z 667.261,A -85,B 0,C 180,E1 -9832.285,E2 -9832.285} C_VEL
LIN {X 0,Y 434.127,Z 651.375,A -85,B 0,C 180,E1 -9832.925,E2 -9832.925} C_VEL
LIN {X 0,Y 434.799,Z 636.699,A -85,B 0,C 180,E1 -9833.328,E2 -9833.328} C_VEL
LIN {X 0,Y 437.13,Z 503.149,A -85,B 0,C 180,E1 -9835.615,E2 -9835.615} C_VEL
LIN {X 0,Y 431.812,Z 475.542,A -85,B 0,C 180,E1 -9836.472,E2 -9836.472} C_VEL
LIN {X 0,Y 430.838,Z 470.934,A -85,B 0,C 180,E1 -9836.641,E2 -9836.641} C_VEL
LIN {X 0,Y 431.363,Z 463.095,A -85,B 0,C 180,E1 -9837.93,E2 -9837.93} C_VEL
LIN {X 0,Y 428.174,Z 449.034,A -85,B 0,C 180,E1 -9840.585,E2 -9840.585} C_VEL
LIN {X 0,Y 425.284,Z 438.137,A -85,B 0,C 180,E1 -9842.797,E2 -9842.797} C_VEL
LIN {X 0,Y 425.281,Z 438.135,A -85,B 0,C 180,E1 -9845.929,E2 -9845.929} C_VEL
LIN {X 0,Y 425.309,Z 438.131,A -85,B 0,C 180,E1 -9849.046,E2 -9849.046} C_VEL
LIN {X 0,Y 425.327,Z 438.124,A -85,B 0,C 180,E1 -9852.645,E2 -9852.645} C_VEL
LIN {X 0,Y 425.289,Z 438.134,A -85,B 0,C 180,E1 -9855.281,E2 -9855.281} C_VEL
LIN {X 0,Y 425.269,Z 438.139,A -85,B 0,C 180,E1 -9858.621,E2 -9858.621} C_VEL
LIN {X 0,Y 425.309,Z 438.13,A -85,B 0,C 180,E1 -9861.103,E2 -9861.103} C_VEL
LIN {X 0,Y 425.294,Z 438.133,A -85,B 0,C 180,E1 -9864.664,E2 -9864.664} C_VEL
LIN {X 0,Y 425.259,Z 438.137,A -85,B 0,C 180,E1 -9868.073,E2 -9868.073} C_VEL
LIN {X 0,Y 425.324,Z 438.127,A -85,B 0,C 180,E1 -9871.368,E2 -9871.368} C_VEL
LIN {X 0,Y 425.289,Z 438.135,A -85,B 0,C 180,E1 -9874.554,E2 -9874.554} C_VEL
LIN {X 0,Y 425.28,Z 438.133,A -85,B 0,C 180,E1 -9877.661,E2 -9877.661} C_VEL
LIN {X 0,Y 425.354,Z 438.127,A -85,B 0,C 180,E1 -9880.704,E2 -9880.704} C_VEL
LIN {X 0,Y 425.381,Z 438.116,A -85,B 0,C 180,E1 -9883.688,E2 -9883.688} C_VEL
LIN {X 0,Y 425.422,Z 438.112,A -85,B 0,C 180,E1 -9887.599,E2 -9887.599} C_VEL
LIN {X 0,Y 425.435,Z 438.112,A -85,B 0,C 180,E1 -9891.45,E2 -9891.45} C_VEL
LIN {X 0,Y 425.547,Z 438.099,A -85,B 0,C 180,E1 -9894.313,E2 -9894.313} C_VEL
LIN {X 0,Y 425.568,Z 438.095,A -85,B 0,C 180,E1 -9898.107,E2 -9898.107} C_VEL
LIN {X 0,Y 425.695,Z 438.084,A -85,B 0,C 180,E1 -9900,E2 -9900} C_VEL
LIN {X 0,Y 425.551,Z 438.101,A -85,B 0,C 180,E1 -9902.84,E2 -9902.84} C_VEL
LIN {X 0,Y 425.524,Z 438.105,A -85,B 0,C 180,E1 -9906.639,E2 -9906.639} C_VEL
LIN {X 0,Y 425.394,Z 438.119,A -85,B 0,C 180,E1 -9909.51,E2 -9909.51} C_VEL
LIN {X 0,Y 425.386,Z 438.12,A -85,B 0,C 180,E1 -9912.904,E2 -9912.904} C_VEL
LIN {X 0,Y 425.363,Z 438.124,A -85,B 0,C 180,E1 -9916.609,E2 -9916.609} C_VEL
LIN {X 0,Y 425.322,Z 438.127,A -85,B 0,C 180,E1 -9919.636,E2 -9919.636} C_VEL
LIN {X 0,Y 425.301,Z 438.132,A -85,B 0,C 180,E1 -9923.366,E2 -9923.366} C_VEL
LIN {X 0,Y 425.343,Z 438.124,A -85,B 0,C 180,E1 -9926.845,E2 -9926.845} C_VEL
LIN {X 0,Y 425.313,Z 438.128,A -85,B 0,C 180,E1 -9929.718,E2 -9929.718} C_VEL
LIN {X 0,Y 425.279,Z 438.134,A -85,B 0,C 180,E1 -9933.049,E2 -9933.049} C_VEL
LIN {X 0,Y 425.281,Z 438.138,A -85,B 0,C 180,E1 -9935.93,E2 -9935.93} C_VEL
LIN {X 0,Y 425.338,Z 438.246,A -85,B 0,C 180,E1 -9938.705,E2 -9938.705} C_VEL
LIN {X 0,Y 428.263,Z 450.07,A -85,B 0,C 180,E1 -9941.262,E2 -9941.262} C_VEL
LIN {X 0,Y 435.592,Z 467.546,A -85,B 0,C 180,E1 -9942.088,E2 -9942.088} C_VEL
LIN {X 0,Y 437.492,Z 476.115,A -85,B 0,C 180,E1 -9942.37,E2 -9942.37} C_VEL
LIN {X 0,Y 435.022,Z 615.018,A -85,B 0,C 180,E1 -9944.76,E2 -9944.76} C_VEL
LIN {X 0,Y 434.42,Z 630.282,A -85,B 0,C 180,E1 -9945.206,E2 -9945.206} C_VEL
LIN {X 0,Y 433.625,Z 644.909,A -85,B 0,C 180,E1 -9945.821,E2 -9945.821} C_VEL
LIN {X 0,Y 432.627,Z 659.87,A -85,B 0,C 180,E1 -9946.66,E2 -9946.66} C_VEL
LIN {X 0,Y 431.513,Z 673.584,A -85,B 0,C 180,E1 -9947.635,E2 -9947.635} C_VEL
LIN {X 0,Y 430.351,Z 687.009,A -85,B 0,C 180,E1 -9948.818,E2 -9948.818} C_VEL
LIN {X 0,Y 429.123,Z 699.444,A -85,B 0,C 180,E1 -9950.152,E2 -9950.152} C_VEL
LIN {X 0,Y 427.999,Z 710.67,A -85,B 0,C 180,E1 -9951.602,E2 -9951.602} C_VEL
LIN {X 0,Y 426.976,Z 720.234,A -85,B 0,C 180,E1 -9953.075,E2 -9953.075} C_VEL
LIN {X 0,Y 426.09,Z 729.282,A -85,B 0,C 180,E1 -9954.741,E2 -9954.741} C_VEL
LIN {X 0,Y 425.476,Z 736.779,A -85,B 0,C 180,E1 -9956.404,E2 -9956.404} C_VEL
LIN {X 0,Y 424.921,Z 742.948,A -85,B 0,C 180,E1 -9958.045,E2 -9958.045} C_VEL
LIN {X 0,Y 424.588,Z 748.333,A -85,B 0,C 180,E1 -9959.803,E2 -9959.803} C_VEL
LIN {X 0,Y 424.287,Z 752.165,A -85,B 0,C 180,E1 -9961.391,E2 -9961.391} C_VEL
LIN {X 0,Y 424.058,Z 755.928,A -85,B 0,C 180,E1 -9963.503,E2 -9963.503} C_VEL
LIN {X 0,Y 423.938,Z 758.345,A -85,B 0,C 180,E1 -9965.756,E2 -9965.756} C_VEL
LIN {X 0,Y 423.936,Z 759.139,A -85,B 0,C 180,E1 -9968.182,E2 -9968.182} C_VEL
LIN {X 0,Y 423.94,Z 758.539,A -85,B 0,C 180,E1 -9969.892,E2 -9969.892} C_VEL
LIN {X 0,Y 423.298,Z 758.043,A -85,B 0,C 180,E1 -9970.681,E2 -9970.681} C_VEL
LIN {X 0,Y 420.517,Z 756.819,A -85,B 0,C 180,E1 -9971.963,E2 -9971.963} C_VEL
LIN {X 0,Y 418.193,Z 755.497,A -85,B 0,C 180,E1 -9972.989,E2 -9972.989} C_VEL
LIN {X 0,Y 417.242,Z 754.249,A -85,B 0,C 180,E1 -9973.775,E2 -9973.775} C_VEL
LIN {X 0,Y 417.189,Z 753.759,A -85,B 0,C 180,E1 -9974.039,E2 -9974.039} C_VEL
LIN {X 0,Y 417.453,Z 749.759,A -85,B 0,C 180,E1 -9975.871,E2 -9975.871} C_VEL
LIN {X 0,Y 417.832,Z 744.031,A -85,B 0,C 180,E1 -9977.873,E2 -9977.873} C_VEL
LIN {X 0,Y 418.441,Z 736.845,A -85,B 0,C 180,E1 -9979.843,E2 -9979.843} C_VEL
LIN {X 0,Y 419.173,Z 729.057,A -85,B 0,C 180,E1 -9981.58,E2 -9981.58} C_VEL
LIN {X 0,Y 420.066,Z 719.894,A -85,B 0,C 180,E1 -9983.275,E2 -9983.275} C_VEL
LIN {X 0,Y 421.045,Z 710.518,A -85,B 0,C 180,E1 -9984.733,E2 -9984.733} C_VEL
LIN {X 0,Y 422.181,Z 699.403,A -85,B 0,C 180,E1 -9986.183,E2 -9986.183} C_VEL
LIN {X 0,Y 423.405,Z 687.235,A -85,B 0,C 180,E1 -9987.503,E2 -9987.503} C_VEL
LIN {X 0,Y 424.682,Z 673.879,A -85,B 0,C 180,E1 -9988.697,E2 -9988.697} C_VEL
LIN {X 0,Y 425.752,Z 660.812,A -85,B 0,C 180,E1 -9989.646,E2 -9989.646} C_VEL
LIN {X 0,Y 426.743,Z 646.556,A -85,B 0,C 180,E1 -9990.472,E2 -9990.472} C_VEL
LIN {X 0,Y 427.588,Z 631.862,A -85,B 0,C 180,E1 -9991.119,E2 -9991.119} C_VEL
LIN {X 0,Y 428.183,Z 616.849,A -85,B 0,C 180,E1 -9991.588,E2 -9991.588} C_VEL
LIN {X 0,Y 428.704,Z 592.82,A -85,B 0,C 180,E1 -9992.041,E2 -9992.041} C_VEL
LIN {X 0,Y 430.655,Z 476.306,A -85,B 0,C 180,E1 -9994.051,E2 -9994.051} C_VEL
LIN {X 0,Y 428.372,Z 467.158,A -85,B 0,C 180,E1 -9994.367,E2 -9994.367} C_VEL
LIN {X 0,Y 420.886,Z 449.533,A -85,B 0,C 180,E1 -9995.21,E2 -9995.21} C_VEL
LIN {X 0,Y 418.453,Z 438.989,A -85,B 0,C 180,E1 -9997.526,E2 -9997.526} C_VEL
LIN {X 0,Y 418.346,Z 438.988,A -85,B 0,C 180,E1 -10000.65,E2 -10000.65} C_VEL
LIN {X 0,Y 418.33,Z 439.001,A -85,B 0,C 180,E1 -10003.604,E2 -10003.604} C_VEL
LIN {X 0,Y 418.317,Z 439.001,A -85,B 0,C 180,E1 -10006.736,E2 -10006.736} C_VEL
LIN {X 0,Y 418.304,Z 439.006,A -85,B 0,C 180,E1 -10009.801,E2 -10009.801} C_VEL
LIN {X 0,Y 418.292,Z 439.002,A -85,B 0,C 180,E1 -10013.781,E2 -10013.781} C_VEL
LIN {X 0,Y 418.314,Z 439.002,A -85,B 0,C 180,E1 -10017.07,E2 -10017.07} C_VEL
LIN {X 0,Y 418.262,Z 439.008,A -85,B 0,C 180,E1 -10020.271,E2 -10020.271} C_VEL
LIN {X 0,Y 418.252,Z 439.007,A -85,B 0,C 180,E1 -10023.677,E2 -10023.677} C_VEL
LIN {X 0,Y 418.249,Z 439.007,A -85,B 0,C 180,E1 -10027.223,E2 -10027.223} C_VEL
LIN {X 0,Y 418.259,Z 439.008,A -85,B 0,C 180,E1 -10029.681,E2 -10029.681} C_VEL
LIN {X 0,Y 418.235,Z 439.006,A -85,B 0,C 180,E1 -10032.321,E2 -10032.321} C_VEL
LIN {X 0,Y 418.24,Z 439.009,A -85,B 0,C 180,E1 -10035.109,E2 -10035.109} C_VEL
LIN {X 0,Y 418.258,Z 439.004,A -85,B 0,C 180,E1 -10037.769,E2 -10037.769} C_VEL
LIN {X 0,Y 418.269,Z 439.005,A -85,B 0,C 180,E1 -10040.617,E2 -10040.617} C_VEL
LIN {X 0,Y 418.248,Z 439.003,A -85,B 0,C 180,E1 -10043.976,E2 -10043.976} C_VEL
LIN {X 0,Y 418.259,Z 439.008,A -85,B 0,C 180,E1 -10047.156,E2 -10047.156} C_VEL
LIN {X 0,Y 418.27,Z 438.997,A -85,B 0,C 180,E1 -10050.895,E2 -10050.895} C_VEL
LIN {X 0,Y 418.272,Z 439.006,A -85,B 0,C 180,E1 -10054.096,E2 -10054.096} C_VEL
LIN {X 0,Y 418.233,Z 439,A -85,B 0,C 180,E1 -10057.263,E2 -10057.263} C_VEL
LIN {X 0,Y 418.284,Z 439.003,A -85,B 0,C 180,E1 -10060.364,E2 -10060.364} C_VEL
LIN {X 0,Y 418.318,Z 438.992,A -85,B 0,C 180,E1 -10063.404,E2 -10063.404} C_VEL
LIN {X 0,Y 418.347,Z 438.996,A -85,B 0,C 180,E1 -10066.999,E2 -10066.999} C_VEL
LIN {X 0,Y 418.341,Z 438.987,A -85,B 0,C 180,E1 -10070.328,E2 -10070.328} C_VEL
LIN {X 0,Y 418.514,Z 438.974,A -85,B 0,C 180,E1 -10072.279,E2 -10072.279} C_VEL
LIN {X 0,Y 418.513,Z 438.975,A -85,B 0,C 180,E1 -10074.217,E2 -10074.217} C_VEL
LIN {X 0,Y 418.542,Z 438.97,A -85,B 0,C 180,E1 -10078.075,E2 -10078.075} C_VEL
LIN {X 0,Y 418.672,Z 438.959,A -85,B 0,C 180,E1 -10080,E2 -10080} C_VEL
LIN {X 0,Y 418.51,Z 438.97,A -85,B 0,C 180,E1 -10082.887,E2 -10082.887} C_VEL
LIN {X 0,Y 418.493,Z 438.974,A -85,B 0,C 180,E1 -10086.751,E2 -10086.751} C_VEL
LIN {X 0,Y 418.4,Z 438.989,A -85,B 0,C 180,E1 -10088.695,E2 -10088.695} C_VEL
LIN {X 0,Y 418.315,Z 438.991,A -85,B 0,C 180,E1 -10091.631,E2 -10091.631} C_VEL
LIN {X 0,Y 418.302,Z 439.001,A -85,B 0,C 180,E1 -10094.597,E2 -10094.597} C_VEL
LIN {X 0,Y 418.288,Z 439,A -85,B 0,C 180,E1 -10097.604,E2 -10097.604} C_VEL
LIN {X 0,Y 418.25,Z 439.007,A -85,B 0,C 180,E1 -10100.663,E2 -10100.663} C_VEL
LIN {X 0,Y 418.288,Z 439.008,A -85,B 0,C 180,E1 -10103.781,E2 -10103.781} C_VEL
LIN {X 0,Y 418.31,Z 439.001,A -85,B 0,C 180,E1 -10107.07,E2 -10107.07} C_VEL
LIN {X 0,Y 418.258,Z 439.007,A -85,B 0,C 180,E1 -10110.271,E2 -10110.271} C_VEL
LIN {X 0,Y 418.248,Z 439.011,A -85,B 0,C 180,E1 -10113.677,E2 -10113.677} C_VEL
LIN {X 0,Y 418.245,Z 439.011,A -85,B 0,C 180,E1 -10117.223,E2 -10117.223} C_VEL
LIN {X 0,Y 418.255,Z 439.012,A -85,B 0,C 180,E1 -10119.681,E2 -10119.681} C_VEL
LIN {X 0,Y 418.23,Z 439.012,A -85,B 0,C 180,E1 -10122.321,E2 -10122.321} C_VEL
LIN {X 0,Y 418.258,Z 439.009,A -85,B 0,C 180,E1 -10125.112,E2 -10125.112} C_VEL
LIN {X 0,Y 418.291,Z 439.007,A -85,B 0,C 180,E1 -10127.773,E2 -10127.773} C_VEL
LIN {X 0,Y 418.253,Z 439.012,A -85,B 0,C 180,E1 -10131.558,E2 -10131.558} C_VEL
LIN {X 0,Y 418.259,Z 439.011,A -85,B 0,C 180,E1 -10135.159,E2 -10135.159} C_VEL
LIN {X 0,Y 418.28,Z 439.166,A -85,B 0,C 180,E1 -10136.989,E2 -10136.989} C_VEL
LIN {X 0,Y 422.213,Z 454.613,A -85,B 0,C 180,E1 -10140.042,E2 -10140.042} C_VEL
LIN {X 0,Y 424.453,Z 464.602,A -85,B 0,C 180,E1 -10141.921,E2 -10141.921} C_VEL
LIN {X 0,Y 424.328,Z 468.855,A -85,B 0,C 180,E1 -10142.637,E2 -10142.637} C_VEL
LIN {X 0,Y 424.083,Z 471.439,A -85,B 0,C 180,E1 -10143.049,E2 -10143.049} C_VEL
LIN {X 0,Y 430.454,Z 504.325,A -85,B 0,C 180,E1 -10144.07,E2 -10144.07} C_VEL
LIN {X 0,Y 428.084,Z 637.54,A -85,B 0,C 180,E1 -10146.379,E2 -10146.379} C_VEL
LIN {X 0,Y 427.349,Z 653.308,A -85,B 0,C 180,E1 -10146.834,E2 -10146.834} C_VEL
LIN {X 0,Y 426.459,Z 668.627,A -85,B 0,C 180,E1 -10147.484,E2 -10147.484} C_VEL
LIN {X 0,Y 425.366,Z 683.19,A -85,B 0,C 180,E1 -10148.304,E2 -10148.304} C_VEL
LIN {X 0,Y 424.202,Z 696.609,A -85,B 0,C 180,E1 -10149.259,E2 -10149.259} C_VEL
LIN {X 0,Y 422.844,Z 710.265,A -85,B 0,C 180,E1 -10150.458,E2 -10150.458} C_VEL
LIN {X 0,Y 421.547,Z 723.266,A -85,B 0,C 180,E1 -10151.86,E2 -10151.86} C_VEL
LIN {X 0,Y 420.538,Z 733.959,A -85,B 0,C 180,E1 -10153.245,E2 -10153.245} C_VEL
LIN {X 0,Y 419.413,Z 744.937,A -85,B 0,C 180,E1 -10154.946,E2 -10154.946} C_VEL
LIN {X 0,Y 418.474,Z 754.759,A -85,B 0,C 180,E1 -10156.8,E2 -10156.8} C_VEL
LIN {X 0,Y 418.075,Z 761.618,A -85,B 0,C 180,E1 -10158.362,E2 -10158.362} C_VEL
LIN {X 0,Y 417.481,Z 768.677,A -85,B 0,C 180,E1 -10160.308,E2 -10160.308} C_VEL
LIN {X 0,Y 417.233,Z 774.229,A -85,B 0,C 180,E1 -10162.255,E2 -10162.255} C_VEL
LIN {X 0,Y 417.064,Z 778.426,A -85,B 0,C 180,E1 -10164.197,E2 -10164.197} C_VEL
LIN {X 0,Y 416.976,Z 781.369,A -85,B 0,C 180,E1 -10166.134,E2 -10166.134} C_VEL
LIN {X 0,Y 417.047,Z 783.127,A -85,B 0,C 180,E1 -10168.068,E2 -10168.068} C_VEL
LIN {X 0,Y 417.001,Z 783.724,A -85,B 0,C 180,E1 -10169.999,E2 -10169.999} C_VEL
LIN {X 0,Y 417.048,Z 783.12,A -85,B 0,C 180,E1 -10171.931,E2 -10171.931} C_VEL
LIN {X 0,Y 416.99,Z 781.362,A -85,B 0,C 180,E1 -10173.865,E2 -10173.865} C_VEL
LIN {X 0,Y 417.069,Z 778.428,A -85,B 0,C 180,E1 -10175.802,E2 -10175.802} C_VEL
LIN {X 0,Y 417.232,Z 774.247,A -85,B 0,C 180,E1 -10177.744,E2 -10177.744} C_VEL
LIN {X 0,Y 417.48,Z 768.709,A -85,B 0,C 180,E1 -10179.691,E2 -10179.691} C_VEL
LIN {X 0,Y 418.078,Z 761.672,A -85,B 0,C 180,E1 -10181.637,E2 -10181.637} C_VEL
LIN {X 0,Y 418.485,Z 754.808,A -85,B 0,C 180,E1 -10183.204,E2 -10183.204} C_VEL
LIN {X 0,Y 419.411,Z 745.067,A -85,B 0,C 180,E1 -10185.053,E2 -10185.053} C_VEL
LIN {X 0,Y 420.53,Z 734.176,A -85,B 0,C 180,E1 -10186.755,E2 -10186.755} C_VEL
LIN {X 0,Y 421.82,Z 722.023,A -85,B 0,C 180,E1 -10188.319,E2 -10188.319} C_VEL
LIN {X 0,Y 422.901,Z 710.691,A -85,B 0,C 180,E1 -10189.538,E2 -10189.538} C_VEL
LIN {X 0,Y 424.224,Z 697.207,A -85,B 0,C 180,E1 -10190.738,E2 -10190.738} C_VEL
LIN {X 0,Y 425.402,Z 683.98,A -85,B 0,C 180,E1 -10191.693,E2 -10191.693} C_VEL
LIN {X 0,Y 426.519,Z 669.359,A -85,B 0,C 180,E1 -10192.536,E2 -10192.536} C_VEL
LIN {X 0,Y 427.441,Z 654.253,A -85,B 0,C 180,E1 -10193.193,E2 -10193.193} C_VEL
LIN {X 0,Y 428.208,Z 639.238,A -85,B 0,C 180,E1 -10193.645,E2 -10193.645} C_VEL
LIN {X 0,Y 428.795,Z 609.887,A -85,B 0,C 180,E1 -10194.188,E2 -10194.188} C_VEL
LIN {X 0,Y 430.734,Z 504.435,A -85,B 0,C 180,E1 -10196.006,E2 -10196.006} C_VEL
LIN {X 0,Y 425.797,Z 478.213,A -85,B 0,C 180,E1 -10196.833,E2 -10196.833} C_VEL
LIN {X 0,Y 424.243,Z 470.653,A -85,B 0,C 180,E1 -10197.114,E2 -10197.114} C_VEL
LIN {X 0,Y 424.562,Z 464.883,A -85,B 0,C 180,E1 -10198.084,E2 -10198.084} C_VEL
LIN {X 0,Y 421.673,Z 452.038,A -85,B 0,C 180,E1 -10200.552,E2 -10200.552} C_VEL
LIN {X 0,Y 418.233,Z 439.013,A -85,B 0,C 180,E1 -10203.213,E2 -10203.213} C_VEL
LIN {X 0,Y 418.245,Z 439.014,A -85,B 0,C 180,E1 -10206.238,E2 -10206.238} C_VEL
LIN {X 0,Y 418.262,Z 439.006,A -85,B 0,C 180,E1 -10209.679,E2 -10209.679} C_VEL
LIN {X 0,Y 418.28,Z 439.004,A -85,B 0,C 180,E1 -10212.329,E2 -10212.329} C_VEL
LIN {X 0,Y 418.246,Z 439.012,A -85,B 0,C 180,E1 -10215.11,E2 -10215.11} C_VEL
LIN {X 0,Y 418.234,Z 439.01,A -85,B 0,C 180,E1 -10217.766,E2 -10217.766} C_VEL
LIN {X 0,Y 418.254,Z 439.013,A -85,B 0,C 180,E1 -10220.618,E2 -10220.618} C_VEL
LIN {X 0,Y 418.24,Z 439.013,A -85,B 0,C 180,E1 -10223.976,E2 -10223.976} C_VEL
LIN {X 0,Y 418.251,Z 439.006,A -85,B 0,C 180,E1 -10227.156,E2 -10227.156} C_VEL
LIN {X 0,Y 418.261,Z 439.009,A -85,B 0,C 180,E1 -10230.895,E2 -10230.895} C_VEL
LIN {X 0,Y 418.264,Z 439.008,A -85,B 0,C 180,E1 -10234.096,E2 -10234.096} C_VEL
LIN {X 0,Y 418.231,Z 439.01,A -85,B 0,C 180,E1 -10237.264,E2 -10237.264} C_VEL
LIN {X 0,Y 418.276,Z 439.006,A -85,B 0,C 180,E1 -10240.364,E2 -10240.364} C_VEL
LIN {X 0,Y 418.309,Z 438.996,A -85,B 0,C 180,E1 -10243.405,E2 -10243.405} C_VEL
LIN {X 0,Y 418.348,Z 438.994,A -85,B 0,C 180,E1 -10246.994,E2 -10246.994} C_VEL
LIN {X 0,Y 418.352,Z 438.995,A -85,B 0,C 180,E1 -10250.329,E2 -10250.329} C_VEL
LIN {X 0,Y 418.486,Z 438.977,A -85,B 0,C 180,E1 -10253.249,E2 -10253.249} C_VEL
LIN {X 0,Y 418.335,Z 438.997,A -85,B 0,C 180,E1 -10255.182,E2 -10255.182} C_VEL
LIN {X 0,Y 418.538,Z 438.971,A -85,B 0,C 180,E1 -10258.076,E2 -10258.076} C_VEL
LIN {X 0,Y 418.665,Z 438.96,A -85,B 0,C 180,E1 -10260,E2 -10260} C_VEL
LIN {X 0,Y 418.505,Z 438.979,A -85,B 0,C 180,E1 -10262.888,E2 -10262.888} C_VEL
LIN {X 0,Y 418.487,Z 438.981,A -85,B 0,C 180,E1 -10266.751,E2 -10266.751} C_VEL
LIN {X 0,Y 418.335,Z 438.999,A -85,B 0,C 180,E1 -10269.672,E2 -10269.672} C_VEL
LIN {X 0,Y 418.339,Z 438.998,A -85,B 0,C 180,E1 -10273.001,E2 -10273.001} C_VEL
LIN {X 0,Y 418.314,Z 439.002,A -85,B 0,C 180,E1 -10276.739,E2 -10276.739} C_VEL
